//     Standard Inputs/MAIN.R2.In_From_HW/BYTE_[59] <-> Module 3 (Default IO)/Std. In (64 Bytes)/Input DWORD 14 @bit 16
//     Standard Inputs/MAIN.R2.In_From_HW/BYTE_[60] <-> Module 3 (Default IO)/Std. In (64 Bytes)/Input DWORD 14 @bit 24
//     Standard Inputs/MAIN.R2.In_From_HW/BYTE_[62] <-> Module 3 (Default IO)/Std. In (64 Bytes)/Input DWORD 15 @bit 8
//     Standard Inputs/MAIN.R2.In_From_HW/BYTE_[63] <-> Module 3 (Default IO)/Std. In (64 Bytes)/Input DWORD 15 @bit 16
//     Standard Inputs/MAIN.R2.In_From_HW/BYTE_[64] <-> Module 3 (Default IO)/Std. In (64 Bytes)/Input DWORD 15 @bit 24
//     Standard Inputs/MAIN.R2.In_From_HW/BYTE_[6] <-> Module 3 (Default IO)/Std. In (64 Bytes)/Input DWORD 1 @bit 8
//     Standard Inputs/MAIN.R2.In_From_HW/BYTE_[7] <-> Module 3 (Default IO)/Std. In (64 Bytes)/Input DWORD 1 @bit 16
//     Standard Inputs/MAIN.R2.In_From_HW/BYTE_[8] <-> Module 3 (Default IO)/Std. In (64 Bytes)/Input DWORD 1 @bit 24
//     Standard Inputs/MAIN.R2.In_From_HW/BYTE_[{1..61 step 4}] <-> Module 3 (Default IO)/Std. In (64 Bytes)/Input DWORD {0..15}  (16 links)
//     Standard Inputs/MAIN.R2.RT02/External_device_not_connected <-> Module 1 (Sync Inputs)/Compact/External device not connected
//     Standard Inputs/MAIN.R2.RT02/FSOE_Inputs_ConnID <-> Module 2 (Safety Data (8 Byte))/Inputs/FSOE/FSOE ConnID
//     Standard Inputs/MAIN.R2.RT02/FSOE_Inputs_Data_0 <-> Module 2 (Safety Data (8 Byte))/Inputs/FSOE/FSOE Data_0
//     Standard Inputs/MAIN.R2.RT02/FSOE_Inputs_Data_1 <-> Module 2 (Safety Data (8 Byte))/Inputs/FSOE/FSOE Data_1
//     Standard Inputs/MAIN.R2.RT02/FSOE_Inputs_Data_2 <-> Module 2 (Safety Data (8 Byte))/Inputs/FSOE/FSOE Data_2
//     Standard Inputs/MAIN.R2.RT02/FSOE_Inputs_Data_3 <-> Module 2 (Safety Data (8 Byte))/Inputs/FSOE/FSOE Data_3
//     Standard Inputs/MAIN.R2.RT02/InfoData/AdsAddr/netId <-> InfoData/AdsAddr/netId
//     Standard Inputs/MAIN.R2.RT02/InfoData/AdsAddr/port <-> InfoData/AdsAddr/port
//     Standard Inputs/MAIN.R2.RT02/InfoData/State <-> InfoData/State
//     Standard Inputs/MAIN.R2.RT02/TxPDO_State <-> Module 1 (Sync Inputs)/Compact/TxPDO state
//     Standard Inputs/MAIN.R2.RT02/TxPDO_Toogle <-> Module 1 (Sync Inputs)/Compact/TxPDO toggle
//     Standard Outputs/MAIN.R2.Out_To_HW/Byte_[10] <-> Module 3 (Default IO)/Std. Out (64 Bytes)/Output DWORD 2 @bit 8
//     Standard Outputs/MAIN.R2.Out_To_HW/Byte_[11] <-> Module 3 (Default IO)/Std. Out (64 Bytes)/Output DWORD 2 @bit 16
//     Standard Outputs/MAIN.R2.Out_To_HW/Byte_[12] <-> Module 3 (Default IO)/Std. Out (64 Bytes)/Output DWORD 2 @bit 24
//     Standard Outputs/MAIN.R2.Out_To_HW/Byte_[14] <-> Module 3 (Default IO)/Std. Out (64 Bytes)/Output DWORD 3 @bit 8
//     Standard Outputs/MAIN.R2.Out_To_HW/Byte_[15] <-> Module 3 (Default IO)/Std. Out (64 Bytes)/Output DWORD 3 @bit 16
//     Standard Outputs/MAIN.R2.Out_To_HW/Byte_[16] <-> Module 3 (Default IO)/Std. Out (64 Bytes)/Output DWORD 3 @bit 24
//     Standard Outputs/MAIN.R2.Out_To_HW/Byte_[18] <-> Module 3 (Default IO)/Std. Out (64 Bytes)/Output DWORD 4 @bit 8
//     Standard Outputs/MAIN.R2.Out_To_HW/Byte_[19] <-> Module 3 (Default IO)/Std. Out (64 Bytes)/Output DWORD 4 @bit 16
//     Standard Outputs/MAIN.R2.Out_To_HW/Byte_[20] <-> Module 3 (Default IO)/Std. Out (64 Bytes)/Output DWORD 4 @bit 24
//     Standard Outputs/MAIN.R2.Out_To_HW/Byte_[22] <-> Module 3 (Default IO)/Std. Out (64 Bytes)/Output DWORD 5 @bit 8
//     Standard Outputs/MAIN.R2.Out_To_HW/Byte_[23] <-> Module 3 (Default IO)/Std. Out (64 Bytes)/Output DWORD 5 @bit 16
//     Standard Outputs/MAIN.R2.Out_To_HW/Byte_[24] <-> Module 3 (Default IO)/Std. Out (64 Bytes)/Output DWORD 5 @bit 24
//     Standard Outputs/MAIN.R2.Out_To_HW/Byte_[26] <-> Module 3 (Default IO)/Std. Out (64 Bytes)/Output DWORD 6 @bit 8
//     Standard Outputs/MAIN.R2.Out_To_HW/Byte_[27] <-> Module 3 (Default IO)/Std. Out (64 Bytes)/Output DWORD 6 @bit 16
//     Standard Outputs/MAIN.R2.Out_To_HW/Byte_[28] <-> Module 3 (Default IO)/Std. Out (64 Bytes)/Output DWORD 6 @bit 24
//     Standard Outputs/MAIN.R2.Out_To_HW/Byte_[2] <-> Module 3 (Default IO)/Std. Out (64 Bytes)/Output DWORD 0 @bit 8
//     Standard Outputs/MAIN.R2.Out_To_HW/Byte_[30] <-> Module 3 (Default IO)/Std. Out (64 Bytes)/Output DWORD 7 @bit 8
//     Standard Outputs/MAIN.R2.Out_To_HW/Byte_[31] <-> Module 3 (Default IO)/Std. Out (64 Bytes)/Output DWORD 7 @bit 16
//     Standard Outputs/MAIN.R2.Out_To_HW/Byte_[32] <-> Module 3 (Default IO)/Std. Out (64 Bytes)/Output DWORD 7 @bit 24
//     Standard Outputs/MAIN.R2.Out_To_HW/Byte_[34] <-> Module 3 (Default IO)/Std. Out (64 Bytes)/Output DWORD 8 @bit 8
//     Standard Outputs/MAIN.R2.Out_To_HW/Byte_[35] <-> Module 3 (Default IO)/Std. Out (64 Bytes)/Output DWORD 8 @bit 16
//     Standard Outputs/MAIN.R2.Out_To_HW/Byte_[36] <-> Module 3 (Default IO)/Std. Out (64 Bytes)/Output DWORD 8 @bit 24
//     Standard Outputs/MAIN.R2.Out_To_HW/Byte_[38] <-> Module 3 (Default IO)/Std. Out (64 Bytes)/Output DWORD 9 @bit 8
//     Standard Outputs/MAIN.R2.Out_To_HW/Byte_[39] <-> Module 3 (Default IO)/Std. Out (64 Bytes)/Output DWORD 9 @bit 16
//     Standard Outputs/MAIN.R2.Out_To_HW/Byte_[3] <-> Module 3 (Default IO)/Std. Out (64 Bytes)/Output DWORD 0 @bit 16
//     Standard Outputs/MAIN.R2.Out_To_HW/Byte_[40] <-> Module 3 (Default IO)/Std. Out (64 Bytes)/Output DWORD 9 @bit 24
//     Standard Outputs/MAIN.R2.Out_To_HW/Byte_[42] <-> Module 3 (Default IO)/Std. Out (64 Bytes)/Output DWORD 10 @bit 8
//     Standard Outputs/MAIN.R2.Out_To_HW/Byte_[43] <-> Module 3 (Default IO)/Std. Out (64 Bytes)/Output DWORD 10 @bit 16
//     Standard Outputs/MAIN.R2.Out_To_HW/Byte_[44] <-> Module 3 (Default IO)/Std. Out (64 Bytes)/Output DWORD 10 @bit 24
//     Standard Outputs/MAIN.R2.Out_To_HW/Byte_[46] <-> Module 3 (Default IO)/Std. Out (64 Bytes)/Output DWORD 11 @bit 8
//     Standard Outputs/MAIN.R2.Out_To_HW/Byte_[47] <-> Module 3 (Default IO)/Std. Out (64 Bytes)/Output DWORD 11 @bit 16
//     Standard Outputs/MAIN.R2.Out_To_HW/Byte_[48] <-> Module 3 (Default IO)/Std. Out (64 Bytes)/Output DWORD 11 @bit 24
//     Standard Outputs/MAIN.R2.Out_To_HW/Byte_[4] <-> Module 3 (Default IO)/Std. Out (64 Bytes)/Output DWORD 0 @bit 24
//     Standard Outputs/MAIN.R2.Out_To_HW/Byte_[50] <-> Module 3 (Default IO)/Std. Out (64 Bytes)/Output DWORD 12 @bit 8
//     Standard Outputs/MAIN.R2.Out_To_HW/Byte_[51] <-> Module 3 (Default IO)/Std. Out (64 Bytes)/Output DWORD 12 @bit 16
//     Standard Outputs/MAIN.R2.Out_To_HW/Byte_[52] <-> Module 3 (Default IO)/Std. Out (64 Bytes)/Output DWORD 12 @bit 24
//     Standard Outputs/MAIN.R2.Out_To_HW/Byte_[54] <-> Module 3 (Default IO)/Std. Out (64 Bytes)/Output DWORD 13 @bit 8
//     Standard Outputs/MAIN.R2.Out_To_HW/Byte_[55] <-> Module 3 (Default IO)/Std. Out (64 Bytes)/Output DWORD 13 @bit 16
//     Standard Outputs/MAIN.R2.Out_To_HW/Byte_[56] <-> Module 3 (Default IO)/Std. Out (64 Bytes)/Output DWORD 13 @bit 24
//     Standard Outputs/MAIN.R2.Out_To_HW/Byte_[58] <-> Module 3 (Default IO)/Std. Out (64 Bytes)/Output DWORD 14 @bit 8
//     Standard Outputs/MAIN.R2.Out_To_HW/Byte_[59] <-> Module 3 (Default IO)/Std. Out (64 Bytes)/Output DWORD 14 @bit 16
//     Standard Outputs/MAIN.R2.Out_To_HW/Byte_[60] <-> Module 3 (Default IO)/Std. Out (64 Bytes)/Output DWORD 14 @bit 24
//     Standard Outputs/MAIN.R2.Out_To_HW/Byte_[62] <-> Module 3 (Default IO)/Std. Out (64 Bytes)/Output DWORD 15 @bit 8
//     Standard Outputs/MAIN.R2.Out_To_HW/Byte_[63] <-> Module 3 (Default IO)/Std. Out (64 Bytes)/Output DWORD 15 @bit 16
//     Standard Outputs/MAIN.R2.Out_To_HW/Byte_[64] <-> Module 3 (Default IO)/Std. Out (64 Bytes)/Output DWORD 15 @bit 24
//     Standard Outputs/MAIN.R2.Out_To_HW/Byte_[6] <-> Module 3 (Default IO)/Std. Out (64 Bytes)/Output DWORD 1 @bit 8
//     Standard Outputs/MAIN.R2.Out_To_HW/Byte_[7] <-> Module 3 (Default IO)/Std. Out (64 Bytes)/Output DWORD 1 @bit 16
//     Standard Outputs/MAIN.R2.Out_To_HW/Byte_[8] <-> Module 3 (Default IO)/Std. Out (64 Bytes)/Output DWORD 1 @bit 24
//     Standard Outputs/MAIN.R2.Out_To_HW/Byte_[{1..61 step 4}] <-> Module 3 (Default IO)/Std. Out (64 Bytes)/Output DWORD {0..15}  (16 links)
//   SODG11_SSCC610_2403701_PLC/SODG11_SSCC610_2403701_PLC Instance <-> EtherCAT Master (EtherCAT)/R2.T01 (EK1100)
//     Standard Inputs/MAIN.R2.T01/InfoData/State <-> InfoData/State
//   SODG11_SSCC610_2403701_PLC/SODG11_SSCC610_2403701_PLC Instance <-> EtherCAT Master (EtherCAT)/R2.T01 (EK1100)/R2.T02 (EL6900)
//     Standard Inputs/MAIN.R2.RT02/FSOE_Outputs_Data_0 @bit 1 <-> StandardInputs/Standard Out Var 14
//     Standard Inputs/MAIN.R2.RT02/FSOE_Outputs_Data_0 @bit 2 <-> StandardInputs/Standard Out Var 15
//     Standard Inputs/MAIN.R2.RT02/FSOE_Outputs_Data_2 @bit 1 <-> StandardInputs/Standard Out Var 18
//     Standard Inputs/MAIN.R2.RT02/FSOE_Outputs_Data_2 @bit 2 <-> StandardInputs/Standard Out Var 19
//     Standard Inputs/MAIN.R2.RT02/FSOE_Outputs_Data_2 @bit 3 <-> StandardInputs/Standard Out Var 20
//     Standard Inputs/MAIN.R2.RT02/FSOE_Outputs_Data_2 <-> StandardInputs/Standard Out Var 17
//     Standard Inputs/MAIN.R2.T02_STAT/Device_Info_Data/Project_CRC <-> Device Info Data/Project CRC
//     Standard Inputs/MAIN.R2.T02_STAT/FBs_FB_ERR <-> StandardInputs/Standard Out Var 16
//     Standard Inputs/MAIN.R2.T02_STAT/FBs_FB_ERR @bit 16 <-> StandardInputs/Standard Out Var 21
//     Standard Inputs/MAIN.R2.T02_STAT/FBs_FB_ERR @bit 29 <-> StandardInputs/Standard Out Var 22
//     Standard Inputs/MAIN.R2.T02_STAT/InfoData/AdsAddr/netId <-> InfoData/AdsAddr/netId
//     Standard Inputs/MAIN.R2.T02_STAT/InfoData/AdsAddr/port <-> InfoData/AdsAddr/port
//     Standard Inputs/MAIN.R2.T02_STAT/InfoData/State <-> InfoData/State
//     Standard Inputs/MAIN.R2.T02_STAT/SGs_COM_ERR @bit 1 <-> StandardInputs/Standard Out Var 12
//     Standard Inputs/MAIN.R2.T02_STAT/SGs_COM_ERR <-> StandardInputs/Standard Out Var 9
//     Standard Inputs/MAIN.R2.T02_STAT/SGs_FB_ERR @bit 1 <-> StandardInputs/Standard Out Var 11
//     Standard Inputs/MAIN.R2.T02_STAT/SGs_FB_ERR <-> StandardInputs/Standard Out Var 8
//     Standard Inputs/MAIN.R2.T02_STAT/SGs_OUT_ERR <-> StandardInputs/Standard Out Var 10
//     Standard Inputs/MAIN.R2.T02_STAT/SGs_OUT_ERR @bit 1 <-> StandardInputs/Standard Out Var 13
//     Standard Outputs/MAIN.R2.T02_CMD/FBs_ControlPowerPB <-> StandardOutputs/Standard In Var 7
//     Standard Outputs/MAIN.R2.T02_CMD/SGs_ERRAck <-> StandardOutputs/Standard In Var 4
//     Standard Outputs/MAIN.R2.T02_CMD/SGs_ERRAck <-> StandardOutputs/Standard In Var 6
//     Standard Outputs/MAIN.R2.T02_CMD/SGs_RUNSTOP <-> StandardOutputs/Standard In Var 3
//     Standard Outputs/MAIN.R2.T02_CMD/SGs_RUNSTOP <-> StandardOutputs/Standard In Var 5
//     Standard Outputs/MAIN.Safety_Zone_Test <-> StandardOutputs/Standard In Var 23
//   SODG11_SSCC610_2403701_PLC/SODG11_SSCC610_2403701_PLC Instance <-> EtherCAT Master (EtherCAT)/R2.T01 (EK1100)/R2.T03 (EL1904)
//     Standard Inputs/MAIN.R2.T03/I <-> Module 1 (FSOES)/TxPDO/FSOE/InputChannel1
//     Standard Inputs/MAIN.R2.T03/I @bit 1 <-> Module 1 (FSOES)/TxPDO/FSOE/InputChannel2
//     Standard Inputs/MAIN.R2.T03/I @bit 2 <-> Module 1 (FSOES)/TxPDO/FSOE/InputChannel3
//     Standard Inputs/MAIN.R2.T03/I @bit 3 <-> Module 1 (FSOES)/TxPDO/FSOE/InputChannel4
//     Standard Inputs/MAIN.R2.T03/InfoData/State <-> InfoData/State
//   SODG11_SSCC610_2403701_PLC/SODG11_SSCC610_2403701_PLC Instance <-> EtherCAT Master (EtherCAT)/R2.T01 (EK1100)/R2.T04 (EK1122)
//     Standard Inputs/MAIN.R2.T04/InfoData/State <-> InfoData/State
//   SODG11_SSCC610_2403701_PLC/SODG11_SSCC610_2403701_PLC Instance <-> EtherCAT Master (EtherCAT)/R2.T01 (EK1100)/R2.T04 (EK1122)/R2.Reamer[1].N01 (EP1008-0002)
//     Standard Inputs/MAIN.R2.Reamer[1].N01/I <-> Channel 1/Input
//     Standard Inputs/MAIN.R2.Reamer[1].N01/I @bit 1 <-> Channel 2/Input
//     Standard Inputs/MAIN.R2.Reamer[1].N01/I @bit 2 <-> Channel 3/Input
//     Standard Inputs/MAIN.R2.Reamer[1].N01/I @bit 3 <-> Channel 4/Input
//     Standard Inputs/MAIN.R2.Reamer[1].N01/I @bit 4 <-> Channel 5/Input
//     Standard Inputs/MAIN.R2.Reamer[1].N01/I @bit 5 <-> Channel 6/Input
//     Standard Inputs/MAIN.R2.Reamer[1].N01/I @bit 6 <-> Channel 7/Input
//     Standard Inputs/MAIN.R2.Reamer[1].N01/I @bit 7 <-> Channel 8/Input
//     Standard Inputs/MAIN.R2.Reamer[1].N01/InfoData/State <-> InfoData/State
//     Standard Inputs/MAIN.R2.Reamer[1].N01/Wc_State <-> WcState/WcState
//   SODG11_SSCC610_2403701_PLC/SODG11_SSCC610_2403701_PLC Instance <-> EtherCAT Master (EtherCAT)/R2.T01 (EK1100)/R2.T04 (EK1122)/R2.Reamer[1].N30 (EP2028-0002)
//     Standard Inputs/MAIN.R2.Reamer[1].N30_STAT/InfoData/State <-> InfoData/State
//     Standard Outputs/MAIN.R2.Reamer[1].N30/Q <-> Channel 1/Output
//     Standard Outputs/MAIN.R2.Reamer[1].N30/Q @bit {1..7} <-> Channel {2..8}/Output  (7 links)
//   SODG11_SSCC610_2403701_PLC/SODG11_SSCC610_2403701_PLC Instance <-> EtherCAT Master (EtherCAT)/R3.RT02 (EL6695-1001)
//     Standard Inputs/MAIN.R3.In_From_HW/BYTE_[10] <-> Module 3 (Default IO)/Std. In (64 Bytes)/Input DWORD 2 @bit 8
//     Standard Inputs/MAIN.R3.In_From_HW/BYTE_[11] <-> Module 3 (Default IO)/Std. In (64 Bytes)/Input DWORD 2 @bit 16
//     Standard Inputs/MAIN.R3.In_From_HW/BYTE_[12] <-> Module 3 (Default IO)/Std. In (64 Bytes)/Input DWORD 2 @bit 24
//     Standard Inputs/MAIN.R3.In_From_HW/BYTE_[14] <-> Module 3 (Default IO)/Std. In (64 Bytes)/Input DWORD 3 @bit 8
//     Standard Inputs/MAIN.R3.In_From_HW/BYTE_[15] <-> Module 3 (Default IO)/Std. In (64 Bytes)/Input DWORD 3 @bit 16
//     Standard Inputs/MAIN.R3.In_From_HW/BYTE_[16] <-> Module 3 (Default IO)/Std. In (64 Bytes)/Input DWORD 3 @bit 24
//     Standard Inputs/MAIN.R3.In_From_HW/BYTE_[18] <-> Module 3 (Default IO)/Std. In (64 Bytes)/Input DWORD 4 @bit 8
//     Standard Inputs/MAIN.R3.In_From_HW/BYTE_[19] <-> Module 3 (Default IO)/Std. In (64 Bytes)/Input DWORD 4 @bit 16
//     Standard Inputs/MAIN.R3.In_From_HW/BYTE_[20] <-> Module 3 (Default IO)/Std. In (64 Bytes)/Input DWORD 4 @bit 24
//     Standard Inputs/MAIN.R3.In_From_HW/BYTE_[22] <-> Module 3 (Default IO)/Std. In (64 Bytes)/Input DWORD 5 @bit 8
//     Standard Inputs/MAIN.R3.In_From_HW/BYTE_[23] <-> Module 3 (Default IO)/Std. In (64 Bytes)/Input DWORD 5 @bit 16
//     Standard Inputs/MAIN.R3.In_From_HW/BYTE_[24] <-> Module 3 (Default IO)/Std. In (64 Bytes)/Input DWORD 5 @bit 24
//     Standard Inputs/MAIN.R3.In_From_HW/BYTE_[26] <-> Module 3 (Default IO)/Std. In (64 Bytes)/Input DWORD 6 @bit 8
//     Standard Inputs/MAIN.R3.In_From_HW/BYTE_[27] <-> Module 3 (Default IO)/Std. In (64 Bytes)/Input DWORD 6 @bit 16
//     Standard Inputs/MAIN.R3.In_From_HW/BYTE_[28] <-> Module 3 (Default IO)/Std. In (64 Bytes)/Input DWORD 6 @bit 24
//     Standard Inputs/MAIN.R3.In_From_HW/BYTE_[2] <-> Module 3 (Default IO)/Std. In (64 Bytes)/Input DWORD 0 @bit 8
//     Standard Inputs/MAIN.R3.In_From_HW/BYTE_[30] <-> Module 3 (Default IO)/Std. In (64 Bytes)/Input DWORD 7 @bit 8
//     Standard Inputs/MAIN.R3.In_From_HW/BYTE_[31] <-> Module 3 (Default IO)/Std. In (64 Bytes)/Input DWORD 7 @bit 16
//     Standard Inputs/MAIN.R3.In_From_HW/BYTE_[32] <-> Module 3 (Default IO)/Std. In (64 Bytes)/Input DWORD 7 @bit 24
//     Standard Inputs/MAIN.R3.In_From_HW/BYTE_[34] <-> Module 3 (Default IO)/Std. In (64 Bytes)/Input DWORD 8 @bit 8
//     Standard Inputs/MAIN.R3.In_From_HW/BYTE_[35] <-> Module 3 (Default IO)/Std. In (64 Bytes)/Input DWORD 8 @bit 16
//     Standard Inputs/MAIN.R3.In_From_HW/BYTE_[36] <-> Module 3 (Default IO)/Std. In (64 Bytes)/Input DWORD 8 @bit 24
//     Standard Inputs/MAIN.R3.In_From_HW/BYTE_[38] <-> Module 3 (Default IO)/Std. In (64 Bytes)/Input DWORD 9 @bit 8
//     Standard Inputs/MAIN.R3.In_From_HW/BYTE_[39] <-> Module 3 (Default IO)/Std. In (64 Bytes)/Input DWORD 9 @bit 16
//     Standard Inputs/MAIN.R3.In_From_HW/BYTE_[3] <-> Module 3 (Default IO)/Std. In (64 Bytes)/Input DWORD 0 @bit 16
//     Standard Inputs/MAIN.R3.In_From_HW/BYTE_[40] <-> Module 3 (Default IO)/Std. In (64 Bytes)/Input DWORD 9 @bit 24
//     Standard Inputs/MAIN.R3.In_From_HW/BYTE_[42] <-> Module 3 (Default IO)/Std. In (64 Bytes)/Input DWORD 10 @bit 8
//     Standard Inputs/MAIN.R3.In_From_HW/BYTE_[43] <-> Module 3 (Default IO)/Std. In (64 Bytes)/Input DWORD 10 @bit 16
//     Standard Inputs/MAIN.R3.In_From_HW/BYTE_[44] <-> Module 3 (Default IO)/Std. In (64 Bytes)/Input DWORD 10 @bit 24
//     Standard Inputs/MAIN.R3.In_From_HW/BYTE_[46] <-> Module 3 (Default IO)/Std. In (64 Bytes)/Input DWORD 11 @bit 8
//     Standard Inputs/MAIN.R3.In_From_HW/BYTE_[47] <-> Module 3 (Default IO)/Std. In (64 Bytes)/Input DWORD 11 @bit 16
//     Standard Inputs/MAIN.R3.In_From_HW/BYTE_[48] <-> Module 3 (Default IO)/Std. In (64 Bytes)/Input DWORD 11 @bit 24
//     Standard Inputs/MAIN.R3.In_From_HW/BYTE_[4] <-> Module 3 (Default IO)/Std. In (64 Bytes)/Input DWORD 0 @bit 24
//     Standard Inputs/MAIN.R3.In_From_HW/BYTE_[50] <-> Module 3 (Default IO)/Std. In (64 Bytes)/Input DWORD 12 @bit 8
//     Standard Inputs/MAIN.R3.In_From_HW/BYTE_[51] <-> Module 3 (Default IO)/Std. In (64 Bytes)/Input DWORD 12 @bit 16
//     Standard Inputs/MAIN.R3.In_From_HW/BYTE_[52] <-> Module 3 (Default IO)/Std. In (64 Bytes)/Input DWORD 12 @bit 24
//     Standard Inputs/MAIN.R3.In_From_HW/BYTE_[54] <-> Module 3 (Default IO)/Std. In (64 Bytes)/Input DWORD 13 @bit 8
//     Standard Inputs/MAIN.R3.In_From_HW/BYTE_[55] <-> Module 3 (Default IO)/Std. In (64 Bytes)/Input DWORD 13 @bit 16
//     Standard Inputs/MAIN.R3.In_From_HW/BYTE_[56] <-> Module 3 (Default IO)/Std. In (64 Bytes)/Input DWORD 13 @bit 24
//     Standard Inputs/MAIN.R3.In_From_HW/BYTE_[58] <-> Module 3 (Default IO)/Std. In (64 Bytes)/Input DWORD 14 @bit 8
//     Standard Inputs/MAIN.R3.In_From_HW/BYTE_[59] <-> Module 3 (Default IO)/Std. In (64 Bytes)/Input DWORD 14 @bit 16
//     Standard Inputs/MAIN.R3.In_From_HW/BYTE_[60] <-> Module 3 (Default IO)/Std. In (64 Bytes)/Input DWORD 14 @bit 24
//     Standard Inputs/MAIN.R3.In_From_HW/BYTE_[62] <-> Module 3 (Default IO)/Std. In (64 Bytes)/Input DWORD 15 @bit 8
//     Standard Inputs/MAIN.R3.In_From_HW/BYTE_[63] <-> Module 3 (Default IO)/Std. In (64 Bytes)/Input DWORD 15 @bit 16
//     Standard Inputs/MAIN.R3.In_From_HW/BYTE_[64] <-> Module 3 (Default IO)/Std. In (64 Bytes)/Input DWORD 15 @bit 24
//     Standard Inputs/MAIN.R3.In_From_HW/BYTE_[6] <-> Module 3 (Default IO)/Std. In (64 Bytes)/Input DWORD 1 @bit 8
//     Standard Inputs/MAIN.R3.In_From_HW/BYTE_[7] <-> Module 3 (Default IO)/Std. In (64 Bytes)/Input DWORD 1 @bit 16
//     Standard Inputs/MAIN.R3.In_From_HW/BYTE_[8] <-> Module 3 (Default IO)/Std. In (64 Bytes)/Input DWORD 1 @bit 24
//     Standard Inputs/MAIN.R3.In_From_HW/BYTE_[{1..61 step 4}] <-> Module 3 (Default IO)/Std. In (64 Bytes)/Input DWORD {0..15}  (16 links)
//     Standard Inputs/MAIN.R3.RT02/External_device_not_connected <-> Module 1 (Sync Inputs)/Compact/External device not connected
//     Standard Inputs/MAIN.R3.RT02/FSOE_Inputs_ConnID <-> Module 2 (Safety Data (8 Byte))/Inputs/FSOE/FSOE ConnID
//     Standard Inputs/MAIN.R3.RT02/FSOE_Inputs_Data_0 <-> Module 2 (Safety Data (8 Byte))/Inputs/FSOE/FSOE Data_0
//     Standard Inputs/MAIN.R3.RT02/FSOE_Inputs_Data_1 <-> Module 2 (Safety Data (8 Byte))/Inputs/FSOE/FSOE Data_1
//     Standard Inputs/MAIN.R3.RT02/FSOE_Inputs_Data_2 <-> Module 2 (Safety Data (8 Byte))/Inputs/FSOE/FSOE Data_2
//     Standard Inputs/MAIN.R3.RT02/FSOE_Inputs_Data_3 <-> Module 2 (Safety Data (8 Byte))/Inputs/FSOE/FSOE Data_3
//     Standard Inputs/MAIN.R3.RT02/InfoData/AdsAddr/netId <-> InfoData/AdsAddr/netId
//     Standard Inputs/MAIN.R3.RT02/InfoData/AdsAddr/port <-> InfoData/AdsAddr/port
//     Standard Inputs/MAIN.R3.RT02/InfoData/State <-> InfoData/State
//     Standard Inputs/MAIN.R3.RT02/TxPDO_State <-> Module 1 (Sync Inputs)/Compact/TxPDO state
//     Standard Inputs/MAIN.R3.RT02/TxPDO_Toogle <-> Module 1 (Sync Inputs)/Compact/TxPDO toggle
//     Standard Outputs/MAIN.R3.Out_To_HW/Byte_[10] <-> Module 3 (Default IO)/Std. Out (64 Bytes)/Output DWORD 2 @bit 8
//     Standard Outputs/MAIN.R3.Out_To_HW/Byte_[11] <-> Module 3 (Default IO)/Std. Out (64 Bytes)/Output DWORD 2 @bit 16
//     Standard Outputs/MAIN.R3.Out_To_HW/Byte_[12] <-> Module 3 (Default IO)/Std. Out (64 Bytes)/Output DWORD 2 @bit 24
//     Standard Outputs/MAIN.R3.Out_To_HW/Byte_[14] <-> Module 3 (Default IO)/Std. Out (64 Bytes)/Output DWORD 3 @bit 8
//     Standard Outputs/MAIN.R3.Out_To_HW/Byte_[15] <-> Module 3 (Default IO)/Std. Out (64 Bytes)/Output DWORD 3 @bit 16
//     Standard Outputs/MAIN.R3.Out_To_HW/Byte_[16] <-> Module 3 (Default IO)/Std. Out (64 Bytes)/Output DWORD 3 @bit 24
//     Standard Outputs/MAIN.R3.Out_To_HW/Byte_[18] <-> Module 3 (Default IO)/Std. Out (64 Bytes)/Output DWORD 4 @bit 8
//     Standard Outputs/MAIN.R3.Out_To_HW/Byte_[19] <-> Module 3 (Default IO)/Std. Out (64 Bytes)/Output DWORD 4 @bit 16
//     Standard Outputs/MAIN.R3.Out_To_HW/Byte_[20] <-> Module 3 (Default IO)/Std. Out (64 Bytes)/Output DWORD 4 @bit 24
//     Standard Outputs/MAIN.R3.Out_To_HW/Byte_[22] <-> Module 3 (Default IO)/Std. Out (64 Bytes)/Output DWORD 5 @bit 8
//     Standard Outputs/MAIN.R3.Out_To_HW/Byte_[23] <-> Module 3 (Default IO)/Std. Out (64 Bytes)/Output DWORD 5 @bit 16
//     Standard Outputs/MAIN.R3.Out_To_HW/Byte_[24] <-> Module 3 (Default IO)/Std. Out (64 Bytes)/Output DWORD 5 @bit 24
//     Standard Outputs/MAIN.R3.Out_To_HW/Byte_[26] <-> Module 3 (Default IO)/Std. Out (64 Bytes)/Output DWORD 6 @bit 8
//     Standard Outputs/MAIN.R3.Out_To_HW/Byte_[27] <-> Module 3 (Default IO)/Std. Out (64 Bytes)/Output DWORD 6 @bit 16
//     Standard Outputs/MAIN.R3.Out_To_HW/Byte_[28] <-> Module 3 (Default IO)/Std. Out (64 Bytes)/Output DWORD 6 @bit 24
//     Standard Outputs/MAIN.R3.Out_To_HW/Byte_[2] <-> Module 3 (Default IO)/Std. Out (64 Bytes)/Output DWORD 0 @bit 8
//     Standard Outputs/MAIN.R3.Out_To_HW/Byte_[30] <-> Module 3 (Default IO)/Std. Out (64 Bytes)/Output DWORD 7 @bit 8
//     Standard Outputs/MAIN.R3.Out_To_HW/Byte_[31] <-> Module 3 (Default IO)/Std. Out (64 Bytes)/Output DWORD 7 @bit 16
//     Standard Outputs/MAIN.R3.Out_To_HW/Byte_[32] <-> Module 3 (Default IO)/Std. Out (64 Bytes)/Output DWORD 7 @bit 24
//     Standard Outputs/MAIN.R3.Out_To_HW/Byte_[34] <-> Module 3 (Default IO)/Std. Out (64 Bytes)/Output DWORD 8 @bit 8
//     Standard Outputs/MAIN.R3.Out_To_HW/Byte_[35] <-> Module 3 (Default IO)/Std. Out (64 Bytes)/Output DWORD 8 @bit 16
//     Standard Outputs/MAIN.R3.Out_To_HW/Byte_[36] <-> Module 3 (Default IO)/Std. Out (64 Bytes)/Output DWORD 8 @bit 24
//     Standard Outputs/MAIN.R3.Out_To_HW/Byte_[38] <-> Module 3 (Default IO)/Std. Out (64 Bytes)/Output DWORD 9 @bit 8
//     Standard Outputs/MAIN.R3.Out_To_HW/Byte_[39] <-> Module 3 (Default IO)/Std. Out (64 Bytes)/Output DWORD 9 @bit 16
//     Standard Outputs/MAIN.R3.Out_To_HW/Byte_[3] <-> Module 3 (Default IO)/Std. Out (64 Bytes)/Output DWORD 0 @bit 16
//     Standard Outputs/MAIN.R3.Out_To_HW/Byte_[40] <-> Module 3 (Default IO)/Std. Out (64 Bytes)/Output DWORD 9 @bit 24
//     Standard Outputs/MAIN.R3.Out_To_HW/Byte_[42] <-> Module 3 (Default IO)/Std. Out (64 Bytes)/Output DWORD 10 @bit 8
//     Standard Outputs/MAIN.R3.Out_To_HW/Byte_[43] <-> Module 3 (Default IO)/Std. Out (64 Bytes)/Output DWORD 10 @bit 16
//     Standard Outputs/MAIN.R3.Out_To_HW/Byte_[44] <-> Module 3 (Default IO)/Std. Out (64 Bytes)/Output DWORD 10 @bit 24
//     Standard Outputs/MAIN.R3.Out_To_HW/Byte_[46] <-> Module 3 (Default IO)/Std. Out (64 Bytes)/Output DWORD 11 @bit 8
//     Standard Outputs/MAIN.R3.Out_To_HW/Byte_[47] <-> Module 3 (Default IO)/Std. Out (64 Bytes)/Output DWORD 11 @bit 16
//     Standard Outputs/MAIN.R3.Out_To_HW/Byte_[48] <-> Module 3 (Default IO)/Std. Out (64 Bytes)/Output DWORD 11 @bit 24
//     Standard Outputs/MAIN.R3.Out_To_HW/Byte_[4] <-> Module 3 (Default IO)/Std. Out (64 Bytes)/Output DWORD 0 @bit 24
//     Standard Outputs/MAIN.R3.Out_To_HW/Byte_[50] <-> Module 3 (Default IO)/Std. Out (64 Bytes)/Output DWORD 12 @bit 8
//     Standard Outputs/MAIN.R3.Out_To_HW/Byte_[51] <-> Module 3 (Default IO)/Std. Out (64 Bytes)/Output DWORD 12 @bit 16
//     Standard Outputs/MAIN.R3.Out_To_HW/Byte_[52] <-> Module 3 (Default IO)/Std. Out (64 Bytes)/Output DWORD 12 @bit 24
//     Standard Outputs/MAIN.R3.Out_To_HW/Byte_[54] <-> Module 3 (Default IO)/Std. Out (64 Bytes)/Output DWORD 13 @bit 8
//     Standard Outputs/MAIN.R3.Out_To_HW/Byte_[55] <-> Module 3 (Default IO)/Std. Out (64 Bytes)/Output DWORD 13 @bit 16
//     Standard Outputs/MAIN.R3.Out_To_HW/Byte_[56] <-> Module 3 (Default IO)/Std. Out (64 Bytes)/Output DWORD 13 @bit 24
//     Standard Outputs/MAIN.R3.Out_To_HW/Byte_[58] <-> Module 3 (Default IO)/Std. Out (64 Bytes)/Output DWORD 14 @bit 8
//     Standard Outputs/MAIN.R3.Out_To_HW/Byte_[59] <-> Module 3 (Default IO)/Std. Out (64 Bytes)/Output DWORD 14 @bit 16
//     Standard Outputs/MAIN.R3.Out_To_HW/Byte_[60] <-> Module 3 (Default IO)/Std. Out (64 Bytes)/Output DWORD 14 @bit 24
//     Standard Outputs/MAIN.R3.Out_To_HW/Byte_[62] <-> Module 3 (Default IO)/Std. Out (64 Bytes)/Output DWORD 15 @bit 8
//     Standard Outputs/MAIN.R3.Out_To_HW/Byte_[63] <-> Module 3 (Default IO)/Std. Out (64 Bytes)/Output DWORD 15 @bit 16
//     Standard Outputs/MAIN.R3.Out_To_HW/Byte_[64] <-> Module 3 (Default IO)/Std. Out (64 Bytes)/Output DWORD 15 @bit 24
//     Standard Outputs/MAIN.R3.Out_To_HW/Byte_[6] <-> Module 3 (Default IO)/Std. Out (64 Bytes)/Output DWORD 1 @bit 8
//     Standard Outputs/MAIN.R3.Out_To_HW/Byte_[7] <-> Module 3 (Default IO)/Std. Out (64 Bytes)/Output DWORD 1 @bit 16
//     Standard Outputs/MAIN.R3.Out_To_HW/Byte_[8] <-> Module 3 (Default IO)/Std. Out (64 Bytes)/Output DWORD 1 @bit 24
//     Standard Outputs/MAIN.R3.Out_To_HW/Byte_[{1..61 step 4}] <-> Module 3 (Default IO)/Std. Out (64 Bytes)/Output DWORD {0..15}  (16 links)
//   SODG11_SSCC610_2403701_PLC/SODG11_SSCC610_2403701_PLC Instance <-> EtherCAT Master (EtherCAT)/R3.T01 (EK1100)
//     Standard Inputs/MAIN.R3.T01/InfoData/State <-> InfoData/State
//   SODG11_SSCC610_2403701_PLC/SODG11_SSCC610_2403701_PLC Instance <-> EtherCAT Master (EtherCAT)/R3.T01 (EK1100)/R3.T02 (EL6900)
//     Standard Inputs/MAIN.R3.RT02/FSOE_Outputs_Data_0 @bit 1 <-> StandardInputs/Standard Out Var 14
//     Standard Inputs/MAIN.R3.RT02/FSOE_Outputs_Data_0 @bit 2 <-> StandardInputs/Standard Out Var 15
//     Standard Inputs/MAIN.R3.RT02/FSOE_Outputs_Data_2 @bit 1 <-> StandardInputs/Standard Out Var 18
//     Standard Inputs/MAIN.R3.RT02/FSOE_Outputs_Data_2 <-> StandardInputs/Standard Out Var 17
//     Standard Inputs/MAIN.R3.T02_STAT/Device_Info_Data/Project_CRC <-> Device Info Data/Project CRC
//     Standard Inputs/MAIN.R3.T02_STAT/FBs_FB_ERR <-> StandardInputs/Standard Out Var 16
//     Standard Inputs/MAIN.R3.T02_STAT/FBs_FB_ERR @bit 16 <-> StandardInputs/Standard Out Var 19
//     Standard Inputs/MAIN.R3.T02_STAT/FBs_FB_ERR @bit 29 <-> StandardInputs/Standard Out Var 20
//     Standard Inputs/MAIN.R3.T02_STAT/InfoData/AdsAddr/netId <-> InfoData/AdsAddr/netId
//     Standard Inputs/MAIN.R3.T02_STAT/InfoData/AdsAddr/port <-> InfoData/AdsAddr/port
//     Standard Inputs/MAIN.R3.T02_STAT/InfoData/State <-> InfoData/State
//     Standard Inputs/MAIN.R3.T02_STAT/SGs_COM_ERR @bit 1 <-> StandardInputs/Standard Out Var 12
//     Standard Inputs/MAIN.R3.T02_STAT/SGs_COM_ERR <-> StandardInputs/Standard Out Var 9
//     Standard Inputs/MAIN.R3.T02_STAT/SGs_FB_ERR @bit 1 <-> StandardInputs/Standard Out Var 11
//     Standard Inputs/MAIN.R3.T02_STAT/SGs_FB_ERR <-> StandardInputs/Standard Out Var 8
//     Standard Inputs/MAIN.R3.T02_STAT/SGs_OUT_ERR <-> StandardInputs/Standard Out Var 10
//     Standard Inputs/MAIN.R3.T02_STAT/SGs_OUT_ERR @bit 1 <-> StandardInputs/Standard Out Var 13
//     Standard Outputs/MAIN.R3.T02_CMD/FBs_ControlPowerPB <-> StandardOutputs/Standard In Var 7
//     Standard Outputs/MAIN.R3.T02_CMD/SGs_ERRAck <-> StandardOutputs/Standard In Var 4
//     Standard Outputs/MAIN.R3.T02_CMD/SGs_ERRAck <-> StandardOutputs/Standard In Var 6
//     Standard Outputs/MAIN.R3.T02_CMD/SGs_RUNSTOP <-> StandardOutputs/Standard In Var 3
//     Standard Outputs/MAIN.R3.T02_CMD/SGs_RUNSTOP <-> StandardOutputs/Standard In Var 5
//     Standard Outputs/MAIN.Safety_Zone_Test <-> StandardOutputs/Standard In Var 21
//   SODG11_SSCC610_2403701_PLC/SODG11_SSCC610_2403701_PLC Instance <-> EtherCAT Master (EtherCAT)/R3.T01 (EK1100)/R3.T03 (EL1904)
//     Standard Inputs/MAIN.R3.T03/I <-> Module 1 (FSOES)/TxPDO/FSOE/InputChannel1
//     Standard Inputs/MAIN.R3.T03/I @bit 1 <-> Module 1 (FSOES)/TxPDO/FSOE/InputChannel2
//     Standard Inputs/MAIN.R3.T03/I @bit 2 <-> Module 1 (FSOES)/TxPDO/FSOE/InputChannel3
//     Standard Inputs/MAIN.R3.T03/I @bit 3 <-> Module 1 (FSOES)/TxPDO/FSOE/InputChannel4
//     Standard Inputs/MAIN.R3.T03/InfoData/State <-> InfoData/State
//   SODG11_SSCC610_2403701_PLC/SODG11_SSCC610_2403701_PLC Instance <-> EtherCAT Master (EtherCAT)/R3.T01 (EK1100)/R3.T04 (EK1122)
//     Standard Inputs/MAIN.R3.T04/InfoData/State <-> InfoData/State
//   SODG11_SSCC610_2403701_PLC/SODG11_SSCC610_2403701_PLC Instance <-> EtherCAT Master (EtherCAT)/R3.T01 (EK1100)/R3.T04 (EK1122)/R3.Reamer[1].N01 (EP1008-0002)
//     Standard Inputs/MAIN.R3.Reamer[1].N01/I <-> Channel 1/Input
//     Standard Inputs/MAIN.R3.Reamer[1].N01/I @bit 1 <-> Channel 2/Input
//     Standard Inputs/MAIN.R3.Reamer[1].N01/I @bit 2 <-> Channel 3/Input
//     Standard Inputs/MAIN.R3.Reamer[1].N01/I @bit 3 <-> Channel 4/Input
//     Standard Inputs/MAIN.R3.Reamer[1].N01/I @bit 4 <-> Channel 5/Input
//     Standard Inputs/MAIN.R3.Reamer[1].N01/I @bit 5 <-> Channel 6/Input
//     Standard Inputs/MAIN.R3.Reamer[1].N01/I @bit 6 <-> Channel 7/Input
//     Standard Inputs/MAIN.R3.Reamer[1].N01/I @bit 7 <-> Channel 8/Input
//     Standard Inputs/MAIN.R3.Reamer[1].N01/InfoData/State <-> InfoData/State
//     Standard Inputs/MAIN.R3.Reamer[1].N01/Wc_State <-> WcState/WcState
//   SODG11_SSCC610_2403701_PLC/SODG11_SSCC610_2403701_PLC Instance <-> EtherCAT Master (EtherCAT)/R3.T01 (EK1100)/R3.T04 (EK1122)/R3.Reamer[1].N30 (EP2028-0002)
//     Standard Inputs/MAIN.R3.Reamer[1].N30_STAT/InfoData/State <-> InfoData/State
//     Standard Outputs/MAIN.R3.Reamer[1].N30/Q <-> Channel 1/Output
//     Standard Outputs/MAIN.R3.Reamer[1].N30/Q @bit {1..7} <-> Channel {2..8}/Output  (7 links)
//   SODG11_SSCC610_2403701_PLC/SODG11_SSCC610_2403701_PLC Instance <-> EtherCAT Master (EtherCAT)/R4.RT02 (EL6695-1001)
//     Standard Inputs/MAIN.R4.In_From_HW/BYTE_[10] <-> Module 3 (Default IO)/Std. In (64 Bytes)/Input DWORD 2 @bit 8
//     Standard Inputs/MAIN.R4.In_From_HW/BYTE_[11] <-> Module 3 (Default IO)/Std. In (64 Bytes)/Input DWORD 2 @bit 16
//     Standard Inputs/MAIN.R4.In_From_HW/BYTE_[12] <-> Module 3 (Default IO)/Std. In (64 Bytes)/Input DWORD 2 @bit 24
//     Standard Inputs/MAIN.R4.In_From_HW/BYTE_[14] <-> Module 3 (Default IO)/Std. In (64 Bytes)/Input DWORD 3 @bit 8
//     Standard Inputs/MAIN.R4.In_From_HW/BYTE_[15] <-> Module 3 (Default IO)/Std. In (64 Bytes)/Input DWORD 3 @bit 16
//     Standard Inputs/MAIN.R4.In_From_HW/BYTE_[16] <-> Module 3 (Default IO)/Std. In (64 Bytes)/Input DWORD 3 @bit 24
//     Standard Inputs/MAIN.R4.In_From_HW/BYTE_[18] <-> Module 3 (Default IO)/Std. In (64 Bytes)/Input DWORD 4 @bit 8
//     Standard Inputs/MAIN.R4.In_From_HW/BYTE_[19] <-> Module 3 (Default IO)/Std. In (64 Bytes)/Input DWORD 4 @bit 16
//     Standard Inputs/MAIN.R4.In_From_HW/BYTE_[20] <-> Module 3 (Default IO)/Std. In (64 Bytes)/Input DWORD 4 @bit 24
//     Standard Inputs/MAIN.R4.In_From_HW/BYTE_[22] <-> Module 3 (Default IO)/Std. In (64 Bytes)/Input DWORD 5 @bit 8
//     Standard Inputs/MAIN.R4.In_From_HW/BYTE_[23] <-> Module 3 (Default IO)/Std. In (64 Bytes)/Input DWORD 5 @bit 16
//     Standard Inputs/MAIN.R4.In_From_HW/BYTE_[24] <-> Module 3 (Default IO)/Std. In (64 Bytes)/Input DWORD 5 @bit 24
//     Standard Inputs/MAIN.R4.In_From_HW/BYTE_[26] <-> Module 3 (Default IO)/Std. In (64 Bytes)/Input DWORD 6 @bit 8
//     Standard Inputs/MAIN.R4.In_From_HW/BYTE_[27] <-> Module 3 (Default IO)/Std. In (64 Bytes)/Input DWORD 6 @bit 16
//     Standard Inputs/MAIN.R4.In_From_HW/BYTE_[28] <-> Module 3 (Default IO)/Std. In (64 Bytes)/Input DWORD 6 @bit 24
//     Standard Inputs/MAIN.R4.In_From_HW/BYTE_[2] <-> Module 3 (Default IO)/Std. In (64 Bytes)/Input DWORD 0 @bit 8
//     Standard Inputs/MAIN.R4.In_From_HW/BYTE_[30] <-> Module 3 (Default IO)/Std. In (64 Bytes)/Input DWORD 7 @bit 8
//     Standard Inputs/MAIN.R4.In_From_HW/BYTE_[31] <-> Module 3 (Default IO)/Std. In (64 Bytes)/Input DWORD 7 @bit 16
//     Standard Inputs/MAIN.R4.In_From_HW/BYTE_[32] <-> Module 3 (Default IO)/Std. In (64 Bytes)/Input DWORD 7 @bit 24
//     Standard Inputs/MAIN.R4.In_From_HW/BYTE_[34] <-> Module 3 (Default IO)/Std. In (64 Bytes)/Input DWORD 8 @bit 8
//     Standard Inputs/MAIN.R4.In_From_HW/BYTE_[35] <-> Module 3 (Default IO)/Std. In (64 Bytes)/Input DWORD 8 @bit 16
//     Standard Inputs/MAIN.R4.In_From_HW/BYTE_[36] <-> Module 3 (Default IO)/Std. In (64 Bytes)/Input DWORD 8 @bit 24
//     Standard Inputs/MAIN.R4.In_From_HW/BYTE_[38] <-> Module 3 (Default IO)/Std. In (64 Bytes)/Input DWORD 9 @bit 8
//     Standard Inputs/MAIN.R4.In_From_HW/BYTE_[39] <-> Module 3 (Default IO)/Std. In (64 Bytes)/Input DWORD 9 @bit 16
//     Standard Inputs/MAIN.R4.In_From_HW/BYTE_[3] <-> Module 3 (Default IO)/Std. In (64 Bytes)/Input DWORD 0 @bit 16
//     Standard Inputs/MAIN.R4.In_From_HW/BYTE_[40] <-> Module 3 (Default IO)/Std. In (64 Bytes)/Input DWORD 9 @bit 24
//     Standard Inputs/MAIN.R4.In_From_HW/BYTE_[42] <-> Module 3 (Default IO)/Std. In (64 Bytes)/Input DWORD 10 @bit 8
//     Standard Inputs/MAIN.R4.In_From_HW/BYTE_[43] <-> Module 3 (Default IO)/Std. In (64 Bytes)/Input DWORD 10 @bit 16
//     Standard Inputs/MAIN.R4.In_From_HW/BYTE_[44] <-> Module 3 (Default IO)/Std. In (64 Bytes)/Input DWORD 10 @bit 24
//     Standard Inputs/MAIN.R4.In_From_HW/BYTE_[46] <-> Module 3 (Default IO)/Std. In (64 Bytes)/Input DWORD 11 @bit 8
//     Standard Inputs/MAIN.R4.In_From_HW/BYTE_[47] <-> Module 3 (Default IO)/Std. In (64 Bytes)/Input DWORD 11 @bit 16
//     Standard Inputs/MAIN.R4.In_From_HW/BYTE_[48] <-> Module 3 (Default IO)/Std. In (64 Bytes)/Input DWORD 11 @bit 24
//     Standard Inputs/MAIN.R4.In_From_HW/BYTE_[4] <-> Module 3 (Default IO)/Std. In (64 Bytes)/Input DWORD 0 @bit 24
//     Standard Inputs/MAIN.R4.In_From_HW/BYTE_[50] <-> Module 3 (Default IO)/Std. In (64 Bytes)/Input DWORD 12 @bit 8
//     Standard Inputs/MAIN.R4.In_From_HW/BYTE_[51] <-> Module 3 (Default IO)/Std. In (64 Bytes)/Input DWORD 12 @bit 16
//     Standard Inputs/MAIN.R4.In_From_HW/BYTE_[52] <-> Module 3 (Default IO)/Std. In (64 Bytes)/Input DWORD 12 @bit 24
//     Standard Inputs/MAIN.R4.In_From_HW/BYTE_[54] <-> Module 3 (Default IO)/Std. In (64 Bytes)/Input DWORD 13 @bit 8
//     Standard Inputs/MAIN.R4.In_From_HW/BYTE_[55] <-> Module 3 (Default IO)/Std. In (64 Bytes)/Input DWORD 13 @bit 16
//     Standard Inputs/MAIN.R4.In_From_HW/BYTE_[56] <-> Module 3 (Default IO)/Std. In (64 Bytes)/Input DWORD 13 @bit 24
//     Standard Inputs/MAIN.R4.In_From_HW/BYTE_[58] <-> Module 3 (Default IO)/Std. In (64 Bytes)/Input DWORD 14 @bit 8
//     Standard Inputs/MAIN.R4.In_From_HW/BYTE_[59] <-> Module 3 (Default IO)/Std. In (64 Bytes)/Input DWORD 14 @bit 16
//     Standard Inputs/MAIN.R4.In_From_HW/BYTE_[60] <-> Module 3 (Default IO)/Std. In (64 Bytes)/Input DWORD 14 @bit 24
//     Standard Inputs/MAIN.R4.In_From_HW/BYTE_[62] <-> Module 3 (Default IO)/Std. In (64 Bytes)/Input DWORD 15 @bit 8
//     Standard Inputs/MAIN.R4.In_From_HW/BYTE_[63] <-> Module 3 (Default IO)/Std. In (64 Bytes)/Input DWORD 15 @bit 16
//     Standard Inputs/MAIN.R4.In_From_HW/BYTE_[64] <-> Module 3 (Default IO)/Std. In (64 Bytes)/Input DWORD 15 @bit 24
//     Standard Inputs/MAIN.R4.In_From_HW/BYTE_[6] <-> Module 3 (Default IO)/Std. In (64 Bytes)/Input DWORD 1 @bit 8
//     Standard Inputs/MAIN.R4.In_From_HW/BYTE_[7] <-> Module 3 (Default IO)/Std. In (64 Bytes)/Input DWORD 1 @bit 16
//     Standard Inputs/MAIN.R4.In_From_HW/BYTE_[8] <-> Module 3 (Default IO)/Std. In (64 Bytes)/Input DWORD 1 @bit 24
//     Standard Inputs/MAIN.R4.In_From_HW/BYTE_[{1..61 step 4}] <-> Module 3 (Default IO)/Std. In (64 Bytes)/Input DWORD {0..15}  (16 links)
//     Standard Inputs/MAIN.R4.RT02/External_device_not_connected <-> Module 1 (Sync Inputs)/Compact/External device not connected
//     Standard Inputs/MAIN.R4.RT02/FSOE_Inputs_ConnID <-> Module 2 (Safety Data (8 Byte))/Inputs/FSOE/FSOE ConnID
//     Standard Inputs/MAIN.R4.RT02/FSOE_Inputs_Data_0 <-> Module 2 (Safety Data (8 Byte))/Inputs/FSOE/FSOE Data_0
//     Standard Inputs/MAIN.R4.RT02/FSOE_Inputs_Data_1 <-> Module 2 (Safety Data (8 Byte))/Inputs/FSOE/FSOE Data_1
//     Standard Inputs/MAIN.R4.RT02/FSOE_Inputs_Data_2 <-> Module 2 (Safety Data (8 Byte))/Inputs/FSOE/FSOE Data_2
//     Standard Inputs/MAIN.R4.RT02/FSOE_Inputs_Data_3 <-> Module 2 (Safety Data (8 Byte))/Inputs/FSOE/FSOE Data_3
//     Standard Inputs/MAIN.R4.RT02/InfoData/AdsAddr/netId <-> InfoData/AdsAddr/netId
//     Standard Inputs/MAIN.R4.RT02/InfoData/AdsAddr/port <-> InfoData/AdsAddr/port
//     Standard Inputs/MAIN.R4.RT02/InfoData/State <-> InfoData/State
//     Standard Inputs/MAIN.R4.RT02/TxPDO_State <-> Module 1 (Sync Inputs)/Compact/TxPDO state
//     Standard Inputs/MAIN.R4.RT02/TxPDO_Toogle <-> Module 1 (Sync Inputs)/Compact/TxPDO toggle
//     Standard Outputs/MAIN.R4.Out_To_HW/Byte_[10] <-> Module 3 (Default IO)/Std. Out (64 Bytes)/Output DWORD 2 @bit 8
//     Standard Outputs/MAIN.R4.Out_To_HW/Byte_[11] <-> Module 3 (Default IO)/Std. Out (64 Bytes)/Output DWORD 2 @bit 16
//     Standard Outputs/MAIN.R4.Out_To_HW/Byte_[12] <-> Module 3 (Default IO)/Std. Out (64 Bytes)/Output DWORD 2 @bit 24
//     Standard Outputs/MAIN.R4.Out_To_HW/Byte_[14] <-> Module 3 (Default IO)/Std. Out (64 Bytes)/Output DWORD 3 @bit 8
//     Standard Outputs/MAIN.R4.Out_To_HW/Byte_[15] <-> Module 3 (Default IO)/Std. Out (64 Bytes)/Output DWORD 3 @bit 16
//     Standard Outputs/MAIN.R4.Out_To_HW/Byte_[16] <-> Module 3 (Default IO)/Std. Out (64 Bytes)/Output DWORD 3 @bit 24
//     Standard Outputs/MAIN.R4.Out_To_HW/Byte_[18] <-> Module 3 (Default IO)/Std. Out (64 Bytes)/Output DWORD 4 @bit 8
//     Standard Outputs/MAIN.R4.Out_To_HW/Byte_[19] <-> Module 3 (Default IO)/Std. Out (64 Bytes)/Output DWORD 4 @bit 16
//     Standard Outputs/MAIN.R4.Out_To_HW/Byte_[20] <-> Module 3 (Default IO)/Std. Out (64 Bytes)/Output DWORD 4 @bit 24
//     Standard Outputs/MAIN.R4.Out_To_HW/Byte_[22] <-> Module 3 (Default IO)/Std. Out (64 Bytes)/Output DWORD 5 @bit 8
//     Standard Outputs/MAIN.R4.Out_To_HW/Byte_[23] <-> Module 3 (Default IO)/Std. Out (64 Bytes)/Output DWORD 5 @bit 16
//     Standard Outputs/MAIN.R4.Out_To_HW/Byte_[24] <-> Module 3 (Default IO)/Std. Out (64 Bytes)/Output DWORD 5 @bit 24
//     Standard Outputs/MAIN.R4.Out_To_HW/Byte_[26] <-> Module 3 (Default IO)/Std. Out (64 Bytes)/Output DWORD 6 @bit 8
//     Standard Outputs/MAIN.R4.Out_To_HW/Byte_[27] <-> Module 3 (Default IO)/Std. Out (64 Bytes)/Output DWORD 6 @bit 16
//     Standard Outputs/MAIN.R4.Out_To_HW/Byte_[28] <-> Module 3 (Default IO)/Std. Out (64 Bytes)/Output DWORD 6 @bit 24
//     Standard Outputs/MAIN.R4.Out_To_HW/Byte_[2] <-> Module 3 (Default IO)/Std. Out (64 Bytes)/Output DWORD 0 @bit 8
//     Standard Outputs/MAIN.R4.Out_To_HW/Byte_[30] <-> Module 3 (Default IO)/Std. Out (64 Bytes)/Output DWORD 7 @bit 8
//     Standard Outputs/MAIN.R4.Out_To_HW/Byte_[31] <-> Module 3 (Default IO)/Std. Out (64 Bytes)/Output DWORD 7 @bit 16
//     Standard Outputs/MAIN.R4.Out_To_HW/Byte_[32] <-> Module 3 (Default IO)/Std. Out (64 Bytes)/Output DWORD 7 @bit 24
//     Standard Outputs/MAIN.R4.Out_To_HW/Byte_[34] <-> Module 3 (Default IO)/Std. Out (64 Bytes)/Output DWORD 8 @bit 8
//     Standard Outputs/MAIN.R4.Out_To_HW/Byte_[35] <-> Module 3 (Default IO)/Std. Out (64 Bytes)/Output DWORD 8 @bit 16
//     Standard Outputs/MAIN.R4.Out_To_HW/Byte_[36] <-> Module 3 (Default IO)/Std. Out (64 Bytes)/Output DWORD 8 @bit 24
//     Standard Outputs/MAIN.R4.Out_To_HW/Byte_[38] <-> Module 3 (Default IO)/Std. Out (64 Bytes)/Output DWORD 9 @bit 8
//     Standard Outputs/MAIN.R4.Out_To_HW/Byte_[39] <-> Module 3 (Default IO)/Std. Out (64 Bytes)/Output DWORD 9 @bit 16
//     Standard Outputs/MAIN.R4.Out_To_HW/Byte_[3] <-> Module 3 (Default IO)/Std. Out (64 Bytes)/Output DWORD 0 @bit 16
//     Standard Outputs/MAIN.R4.Out_To_HW/Byte_[40] <-> Module 3 (Default IO)/Std. Out (64 Bytes)/Output DWORD 9 @bit 24
//     Standard Outputs/MAIN.R4.Out_To_HW/Byte_[42] <-> Module 3 (Default IO)/Std. Out (64 Bytes)/Output DWORD 10 @bit 8
//     Standard Outputs/MAIN.R4.Out_To_HW/Byte_[43] <-> Module 3 (Default IO)/Std. Out (64 Bytes)/Output DWORD 10 @bit 16
//     Standard Outputs/MAIN.R4.Out_To_HW/Byte_[44] <-> Module 3 (Default IO)/Std. Out (64 Bytes)/Output DWORD 10 @bit 24
//     Standard Outputs/MAIN.R4.Out_To_HW/Byte_[46] <-> Module 3 (Default IO)/Std. Out (64 Bytes)/Output DWORD 11 @bit 8
//     Standard Outputs/MAIN.R4.Out_To_HW/Byte_[47] <-> Module 3 (Default IO)/Std. Out (64 Bytes)/Output DWORD 11 @bit 16
//     Standard Outputs/MAIN.R4.Out_To_HW/Byte_[48] <-> Module 3 (Default IO)/Std. Out (64 Bytes)/Output DWORD 11 @bit 24
//     Standard Outputs/MAIN.R4.Out_To_HW/Byte_[4] <-> Module 3 (Default IO)/Std. Out (64 Bytes)/Output DWORD 0 @bit 24
//     Standard Outputs/MAIN.R4.Out_To_HW/Byte_[50] <-> Module 3 (Default IO)/Std. Out (64 Bytes)/Output DWORD 12 @bit 8
//     Standard Outputs/MAIN.R4.Out_To_HW/Byte_[51] <-> Module 3 (Default IO)/Std. Out (64 Bytes)/Output DWORD 12 @bit 16
//     Standard Outputs/MAIN.R4.Out_To_HW/Byte_[52] <-> Module 3 (Default IO)/Std. Out (64 Bytes)/Output DWORD 12 @bit 24
//     Standard Outputs/MAIN.R4.Out_To_HW/Byte_[54] <-> Module 3 (Default IO)/Std. Out (64 Bytes)/Output DWORD 13 @bit 8
//     Standard Outputs/MAIN.R4.Out_To_HW/Byte_[55] <-> Module 3 (Default IO)/Std. Out (64 Bytes)/Output DWORD 13 @bit 16
//     Standard Outputs/MAIN.R4.Out_To_HW/Byte_[56] <-> Module 3 (Default IO)/Std. Out (64 Bytes)/Output DWORD 13 @bit 24
//     Standard Outputs/MAIN.R4.Out_To_HW/Byte_[58] <-> Module 3 (Default IO)/Std. Out (64 Bytes)/Output DWORD 14 @bit 8
//     Standard Outputs/MAIN.R4.Out_To_HW/Byte_[59] <-> Module 3 (Default IO)/Std. Out (64 Bytes)/Output DWORD 14 @bit 16
//     Standard Outputs/MAIN.R4.Out_To_HW/Byte_[60] <-> Module 3 (Default IO)/Std. Out (64 Bytes)/Output DWORD 14 @bit 24
//     Standard Outputs/MAIN.R4.Out_To_HW/Byte_[62] <-> Module 3 (Default IO)/Std. Out (64 Bytes)/Output DWORD 15 @bit 8
//     Standard Outputs/MAIN.R4.Out_To_HW/Byte_[63] <-> Module 3 (Default IO)/Std. Out (64 Bytes)/Output DWORD 15 @bit 16
//     Standard Outputs/MAIN.R4.Out_To_HW/Byte_[64] <-> Module 3 (Default IO)/Std. Out (64 Bytes)/Output DWORD 15 @bit 24
//     Standard Outputs/MAIN.R4.Out_To_HW/Byte_[6] <-> Module 3 (Default IO)/Std. Out (64 Bytes)/Output DWORD 1 @bit 8
//     Standard Outputs/MAIN.R4.Out_To_HW/Byte_[7] <-> Module 3 (Default IO)/Std. Out (64 Bytes)/Output DWORD 1 @bit 16
//     Standard Outputs/MAIN.R4.Out_To_HW/Byte_[8] <-> Module 3 (Default IO)/Std. Out (64 Bytes)/Output DWORD 1 @bit 24
//     Standard Outputs/MAIN.R4.Out_To_HW/Byte_[{1..61 step 4}] <-> Module 3 (Default IO)/Std. Out (64 Bytes)/Output DWORD {0..15}  (16 links)
//   SODG11_SSCC610_2403701_PLC/SODG11_SSCC610_2403701_PLC Instance <-> EtherCAT Master (EtherCAT)/R4.T01 (EK1100)
//     Standard Inputs/MAIN.R4.T01/InfoData/State <-> InfoData/State
//   SODG11_SSCC610_2403701_PLC/SODG11_SSCC610_2403701_PLC Instance <-> EtherCAT Master (EtherCAT)/R4.T01 (EK1100)/R4.T02 (EL6900)
//     Standard Inputs/MAIN.R4.RT02/FSOE_Outputs_Data_0 @bit 1 <-> StandardInputs/Standard Out Var 14
//     Standard Inputs/MAIN.R4.RT02/FSOE_Outputs_Data_0 @bit 2 <-> StandardInputs/Standard Out Var 15
//     Standard Inputs/MAIN.R4.RT02/FSOE_Outputs_Data_2 @bit 1 <-> StandardInputs/Standard Out Var 18
//     Standard Inputs/MAIN.R4.RT02/FSOE_Outputs_Data_2 <-> StandardInputs/Standard Out Var 17
//     Standard Inputs/MAIN.R4.T02_STAT/Device_Info_Data/Project_CRC <-> Device Info Data/Project CRC
//     Standard Inputs/MAIN.R4.T02_STAT/FBs_FB_ERR <-> StandardInputs/Standard Out Var 16
//     Standard Inputs/MAIN.R4.T02_STAT/FBs_FB_ERR @bit 16 <-> StandardInputs/Standard Out Var 19
//     Standard Inputs/MAIN.R4.T02_STAT/FBs_FB_ERR @bit 29 <-> StandardInputs/Standard Out Var 20
//     Standard Inputs/MAIN.R4.T02_STAT/InfoData/AdsAddr/netId <-> InfoData/AdsAddr/netId
//     Standard Inputs/MAIN.R4.T02_STAT/InfoData/AdsAddr/port <-> InfoData/AdsAddr/port
//     Standard Inputs/MAIN.R4.T02_STAT/InfoData/State <-> InfoData/State
//     Standard Inputs/MAIN.R4.T02_STAT/SGs_COM_ERR @bit 1 <-> StandardInputs/Standard Out Var 12
//     Standard Inputs/MAIN.R4.T02_STAT/SGs_COM_ERR <-> StandardInputs/Standard Out Var 9
//     Standard Inputs/MAIN.R4.T02_STAT/SGs_FB_ERR @bit 1 <-> StandardInputs/Standard Out Var 11
//     Standard Inputs/MAIN.R4.T02_STAT/SGs_FB_ERR <-> StandardInputs/Standard Out Var 8
//     Standard Inputs/MAIN.R4.T02_STAT/SGs_OUT_ERR <-> StandardInputs/Standard Out Var 10
//     Standard Inputs/MAIN.R4.T02_STAT/SGs_OUT_ERR @bit 1 <-> StandardInputs/Standard Out Var 13
//     Standard Outputs/MAIN.R4.T02_CMD/FBs_ControlPowerPB <-> StandardOutputs/Standard In Var 7
//     Standard Outputs/MAIN.R4.T02_CMD/SGs_ERRAck <-> StandardOutputs/Standard In Var 4
//     Standard Outputs/MAIN.R4.T02_CMD/SGs_ERRAck <-> StandardOutputs/Standard In Var 6
//     Standard Outputs/MAIN.R4.T02_CMD/SGs_RUNSTOP <-> StandardOutputs/Standard In Var 3
//     Standard Outputs/MAIN.R4.T02_CMD/SGs_RUNSTOP <-> StandardOutputs/Standard In Var 5
//     Standard Outputs/MAIN.Safety_Zone_Test <-> StandardOutputs/Standard In Var 21
//   SODG11_SSCC610_2403701_PLC/SODG11_SSCC610_2403701_PLC Instance <-> EtherCAT Master (EtherCAT)/R4.T01 (EK1100)/R4.T03 (EL1904)
//     Standard Inputs/MAIN.R4.T03/I <-> Module 1 (FSOES)/TxPDO/FSOE/InputChannel1
//     Standard Inputs/MAIN.R4.T03/I @bit 1 <-> Module 1 (FSOES)/TxPDO/FSOE/InputChannel2
//     Standard Inputs/MAIN.R4.T03/I @bit 2 <-> Module 1 (FSOES)/TxPDO/FSOE/InputChannel3
//     Standard Inputs/MAIN.R4.T03/I @bit 3 <-> Module 1 (FSOES)/TxPDO/FSOE/InputChannel4
//     Standard Inputs/MAIN.R4.T03/InfoData/State <-> InfoData/State
//   SODG11_SSCC610_2403701_PLC/SODG11_SSCC610_2403701_PLC Instance <-> EtherCAT Master (EtherCAT)/R4.T01 (EK1100)/R4.T04 (EK1122)
//     Standard Inputs/MAIN.R4.T04/InfoData/State <-> InfoData/State
//   SODG11_SSCC610_2403701_PLC/SODG11_SSCC610_2403701_PLC Instance <-> EtherCAT Master (EtherCAT)/R4.T01 (EK1100)/R4.T04 (EK1122)/EOAT04.N01 (EP1008-0002)
//     Standard Inputs/EOAT04.N01/I <-> Channel 1/Input
//     Standard Inputs/EOAT04.N01/I @bit 1 <-> Channel 2/Input
//     Standard Inputs/EOAT04.N01/I @bit 2 <-> Channel 3/Input
//     Standard Inputs/EOAT04.N01/I @bit 3 <-> Channel 4/Input
//     Standard Inputs/EOAT04.N01/I @bit 4 <-> Channel 5/Input
//     Standard Inputs/EOAT04.N01/I @bit 5 <-> Channel 6/Input
//     Standard Inputs/EOAT04.N01/I @bit 6 <-> Channel 7/Input
//     Standard Inputs/EOAT04.N01/I @bit 7 <-> Channel 8/Input
//     Standard Inputs/EOAT04.N01/InfoData/State <-> InfoData/State
//     Standard Inputs/EOAT04.N01/Wc_State <-> WcState/WcState
//   SODG11_SSCC610_2403701_PLC/SODG11_SSCC610_2403701_PLC Instance <-> EtherCAT Master (EtherCAT)/R4.T01 (EK1100)/R4.T04 (EK1122)/EOAT04.N02 (EP1008-0002)
//     Standard Inputs/EOAT04.N02/I <-> Channel 1/Input
//     Standard Inputs/EOAT04.N02/I @bit 1 <-> Channel 2/Input
//     Standard Inputs/EOAT04.N02/I @bit 2 <-> Channel 3/Input
//     Standard Inputs/EOAT04.N02/I @bit 3 <-> Channel 4/Input
//     Standard Inputs/EOAT04.N02/I @bit 4 <-> Channel 5/Input
//     Standard Inputs/EOAT04.N02/I @bit 5 <-> Channel 6/Input
//     Standard Inputs/EOAT04.N02/I @bit 6 <-> Channel 7/Input
//     Standard Inputs/EOAT04.N02/I @bit 7 <-> Channel 8/Input
//     Standard Inputs/EOAT04.N02/InfoData/State <-> InfoData/State
//     Standard Inputs/EOAT04.N02/Wc_State <-> WcState/WcState
//   SODG11_SSCC610_2403701_PLC/SODG11_SSCC610_2403701_PLC Instance <-> EtherCAT Master (EtherCAT)/R4.T01 (EK1100)/R4.T04 (EK1122)/EOAT04.N03 (EP1008-0002)
//     Standard Inputs/EOAT04.N03/I <-> Channel 1/Input
//     Standard Inputs/EOAT04.N03/I @bit 1 <-> Channel 2/Input
//     Standard Inputs/EOAT04.N03/I @bit 2 <-> Channel 3/Input
//     Standard Inputs/EOAT04.N03/I @bit 3 <-> Channel 4/Input
//     Standard Inputs/EOAT04.N03/I @bit 4 <-> Channel 5/Input
//     Standard Inputs/EOAT04.N03/I @bit 5 <-> Channel 6/Input
//     Standard Inputs/EOAT04.N03/I @bit 6 <-> Channel 7/Input
//     Standard Inputs/EOAT04.N03/I @bit 7 <-> Channel 8/Input
//     Standard Inputs/EOAT04.N03/InfoData/State <-> InfoData/State
//     Standard Inputs/EOAT04.N03/Wc_State <-> WcState/WcState
//   SODG11_SSCC610_2403701_PLC/SODG11_SSCC610_2403701_PLC Instance <-> EtherCAT Master (EtherCAT)/R4.T01 (EK1100)/R4.T04 (EK1122)/EOAT04.N04 (EP1008-0002)
//     Standard Inputs/EOAT04.N04/I <-> Channel 1/Input
//     Standard Inputs/EOAT04.N04/I @bit 1 <-> Channel 2/Input
//     Standard Inputs/EOAT04.N04/I @bit 2 <-> Channel 3/Input
//     Standard Inputs/EOAT04.N04/I @bit 3 <-> Channel 4/Input
//     Standard Inputs/EOAT04.N04/I @bit 4 <-> Channel 5/Input
//     Standard Inputs/EOAT04.N04/I @bit 5 <-> Channel 6/Input
//     Standard Inputs/EOAT04.N04/I @bit 6 <-> Channel 7/Input
//     Standard Inputs/EOAT04.N04/I @bit 7 <-> Channel 8/Input
//     Standard Inputs/EOAT04.N04/InfoData/State <-> InfoData/State
//     Standard Inputs/EOAT04.N04/Wc_State <-> WcState/WcState
//   SODG11_SSCC610_2403701_PLC/SODG11_SSCC610_2403701_PLC Instance <-> EtherCAT Master (EtherCAT)/R4.T01 (EK1100)/R4.T04 (EK1122)/EOAT04.N100 (EX260-SEC1)
//     Standard Inputs/EOAT04.N100_STAT/InfoData/State <-> InfoData/State
//     Standard Outputs/EOAT04.N100/Q <-> Byte 0/Output
//     Standard Outputs/EOAT04.N100/Q @bit 8 <-> Byte 1/Output
//     Standard Outputs/EOAT04.N100/Q @bit 16 <-> Byte 2/Output
//     Standard Outputs/EOAT04.N100/Q @bit 24 <-> Byte 3/Output
//   SODG11_SSCC610_2403701_PLC/SODG11_SSCC610_2403701_PLC Instance <-> EtherCAT Master (EtherCAT)/R5.RT02 (EL6695-1001)
//     Standard Inputs/MAIN.R5.In_From_HW/BYTE_[10] <-> Module 3 (Default IO)/Std. In (64 Bytes)/Input DWORD 2 @bit 8
//     Standard Inputs/MAIN.R5.In_From_HW/BYTE_[11] <-> Module 3 (Default IO)/Std. In (64 Bytes)/Input DWORD 2 @bit 16
//     Standard Inputs/MAIN.R5.In_From_HW/BYTE_[12] <-> Module 3 (Default IO)/Std. In (64 Bytes)/Input DWORD 2 @bit 24
//     Standard Inputs/MAIN.R5.In_From_HW/BYTE_[14] <-> Module 3 (Default IO)/Std. In (64 Bytes)/Input DWORD 3 @bit 8
//     Standard Inputs/MAIN.R5.In_From_HW/BYTE_[15] <-> Module 3 (Default IO)/Std. In (64 Bytes)/Input DWORD 3 @bit 16
//     Standard Inputs/MAIN.R5.In_From_HW/BYTE_[16] <-> Module 3 (Default IO)/Std. In (64 Bytes)/Input DWORD 3 @bit 24
//     Standard Inputs/MAIN.R5.In_From_HW/BYTE_[18] <-> Module 3 (Default IO)/Std. In (64 Bytes)/Input DWORD 4 @bit 8
//     Standard Inputs/MAIN.R5.In_From_HW/BYTE_[19] <-> Module 3 (Default IO)/Std. In (64 Bytes)/Input DWORD 4 @bit 16
//     Standard Inputs/MAIN.R5.In_From_HW/BYTE_[20] <-> Module 3 (Default IO)/Std. In (64 Bytes)/Input DWORD 4 @bit 24
//     Standard Inputs/MAIN.R5.In_From_HW/BYTE_[22] <-> Module 3 (Default IO)/Std. In (64 Bytes)/Input DWORD 5 @bit 8
//     Standard Inputs/MAIN.R5.In_From_HW/BYTE_[23] <-> Module 3 (Default IO)/Std. In (64 Bytes)/Input DWORD 5 @bit 16
//     Standard Inputs/MAIN.R5.In_From_HW/BYTE_[24] <-> Module 3 (Default IO)/Std. In (64 Bytes)/Input DWORD 5 @bit 24
//     Standard Inputs/MAIN.R5.In_From_HW/BYTE_[26] <-> Module 3 (Default IO)/Std. In (64 Bytes)/Input DWORD 6 @bit 8
//     Standard Inputs/MAIN.R5.In_From_HW/BYTE_[27] <-> Module 3 (Default IO)/Std. In (64 Bytes)/Input DWORD 6 @bit 16
//     Standard Inputs/MAIN.R5.In_From_HW/BYTE_[28] <-> Module 3 (Default IO)/Std. In (64 Bytes)/Input DWORD 6 @bit 24
//     Standard Inputs/MAIN.R5.In_From_HW/BYTE_[2] <-> Module 3 (Default IO)/Std. In (64 Bytes)/Input DWORD 0 @bit 8
//     Standard Inputs/MAIN.R5.In_From_HW/BYTE_[30] <-> Module 3 (Default IO)/Std. In (64 Bytes)/Input DWORD 7 @bit 8
//     Standard Inputs/MAIN.R5.In_From_HW/BYTE_[31] <-> Module 3 (Default IO)/Std. In (64 Bytes)/Input DWORD 7 @bit 16
//     Standard Inputs/MAIN.R5.In_From_HW/BYTE_[32] <-> Module 3 (Default IO)/Std. In (64 Bytes)/Input DWORD 7 @bit 24
//     Standard Inputs/MAIN.R5.In_From_HW/BYTE_[34] <-> Module 3 (Default IO)/Std. In (64 Bytes)/Input DWORD 8 @bit 8
//     Standard Inputs/MAIN.R5.In_From_HW/BYTE_[35] <-> Module 3 (Default IO)/Std. In (64 Bytes)/Input DWORD 8 @bit 16
//     Standard Inputs/MAIN.R5.In_From_HW/BYTE_[36] <-> Module 3 (Default IO)/Std. In (64 Bytes)/Input DWORD 8 @bit 24
//     Standard Inputs/MAIN.R5.In_From_HW/BYTE_[38] <-> Module 3 (Default IO)/Std. In (64 Bytes)/Input DWORD 9 @bit 8
//     Standard Inputs/MAIN.R5.In_From_HW/BYTE_[39] <-> Module 3 (Default IO)/Std. In (64 Bytes)/Input DWORD 9 @bit 16
//     Standard Inputs/MAIN.R5.In_From_HW/BYTE_[3] <-> Module 3 (Default IO)/Std. In (64 Bytes)/Input DWORD 0 @bit 16
//     Standard Inputs/MAIN.R5.In_From_HW/BYTE_[40] <-> Module 3 (Default IO)/Std. In (64 Bytes)/Input DWORD 9 @bit 24
//     Standard Inputs/MAIN.R5.In_From_HW/BYTE_[42] <-> Module 3 (Default IO)/Std. In (64 Bytes)/Input DWORD 10 @bit 8
//     Standard Inputs/MAIN.R5.In_From_HW/BYTE_[43] <-> Module 3 (Default IO)/Std. In (64 Bytes)/Input DWORD 10 @bit 16
//     Standard Inputs/MAIN.R5.In_From_HW/BYTE_[44] <-> Module 3 (Default IO)/Std. In (64 Bytes)/Input DWORD 10 @bit 24
//     Standard Inputs/MAIN.R5.In_From_HW/BYTE_[46] <-> Module 3 (Default IO)/Std. In (64 Bytes)/Input DWORD 11 @bit 8
//     Standard Inputs/MAIN.R5.In_From_HW/BYTE_[47] <-> Module 3 (Default IO)/Std. In (64 Bytes)/Input DWORD 11 @bit 16
//     Standard Inputs/MAIN.R5.In_From_HW/BYTE_[48] <-> Module 3 (Default IO)/Std. In (64 Bytes)/Input DWORD 11 @bit 24
//     Standard Inputs/MAIN.R5.In_From_HW/BYTE_[4] <-> Module 3 (Default IO)/Std. In (64 Bytes)/Input DWORD 0 @bit 24
//     Standard Inputs/MAIN.R5.In_From_HW/BYTE_[50] <-> Module 3 (Default IO)/Std. In (64 Bytes)/Input DWORD 12 @bit 8
//     Standard Inputs/MAIN.R5.In_From_HW/BYTE_[51] <-> Module 3 (Default IO)/Std. In (64 Bytes)/Input DWORD 12 @bit 16
//     Standard Inputs/MAIN.R5.In_From_HW/BYTE_[52] <-> Module 3 (Default IO)/Std. In (64 Bytes)/Input DWORD 12 @bit 24
//     Standard Inputs/MAIN.R5.In_From_HW/BYTE_[54] <-> Module 3 (Default IO)/Std. In (64 Bytes)/Input DWORD 13 @bit 8
//     Standard Inputs/MAIN.R5.In_From_HW/BYTE_[55] <-> Module 3 (Default IO)/Std. In (64 Bytes)/Input DWORD 13 @bit 16
//     Standard Inputs/MAIN.R5.In_From_HW/BYTE_[56] <-> Module 3 (Default IO)/Std. In (64 Bytes)/Input DWORD 13 @bit 24
//     Standard Inputs/MAIN.R5.In_From_HW/BYTE_[58] <-> Module 3 (Default IO)/Std. In (64 Bytes)/Input DWORD 14 @bit 8
//     Standard Inputs/MAIN.R5.In_From_HW/BYTE_[59] <-> Module 3 (Default IO)/Std. In (64 Bytes)/Input DWORD 14 @bit 16
//     Standard Inputs/MAIN.R5.In_From_HW/BYTE_[60] <-> Module 3 (Default IO)/Std. In (64 Bytes)/Input DWORD 14 @bit 24
//     Standard Inputs/MAIN.R5.In_From_HW/BYTE_[62] <-> Module 3 (Default IO)/Std. In (64 Bytes)/Input DWORD 15 @bit 8
//     Standard Inputs/MAIN.R5.In_From_HW/BYTE_[63] <-> Module 3 (Default IO)/Std. In (64 Bytes)/Input DWORD 15 @bit 16
//     Standard Inputs/MAIN.R5.In_From_HW/BYTE_[64] <-> Module 3 (Default IO)/Std. In (64 Bytes)/Input DWORD 15 @bit 24
//     Standard Inputs/MAIN.R5.In_From_HW/BYTE_[6] <-> Module 3 (Default IO)/Std. In (64 Bytes)/Input DWORD 1 @bit 8
//     Standard Inputs/MAIN.R5.In_From_HW/BYTE_[7] <-> Module 3 (Default IO)/Std. In (64 Bytes)/Input DWORD 1 @bit 16
//     Standard Inputs/MAIN.R5.In_From_HW/BYTE_[8] <-> Module 3 (Default IO)/Std. In (64 Bytes)/Input DWORD 1 @bit 24
//     Standard Inputs/MAIN.R5.In_From_HW/BYTE_[{1..61 step 4}] <-> Module 3 (Default IO)/Std. In (64 Bytes)/Input DWORD {0..15}  (16 links)
//     Standard Inputs/MAIN.R5.RT02/External_device_not_connected <-> Module 1 (Sync Inputs)/Compact/External device not connected
//     Standard Inputs/MAIN.R5.RT02/FSOE_Inputs_ConnID <-> Module 2 (Safety Data (8 Byte))/Inputs/FSOE/FSOE ConnID
//     Standard Inputs/MAIN.R5.RT02/FSOE_Inputs_Data_0 <-> Module 2 (Safety Data (8 Byte))/Inputs/FSOE/FSOE Data_0
//     Standard Inputs/MAIN.R5.RT02/FSOE_Inputs_Data_1 <-> Module 2 (Safety Data (8 Byte))/Inputs/FSOE/FSOE Data_1
//     Standard Inputs/MAIN.R5.RT02/FSOE_Inputs_Data_2 <-> Module 2 (Safety Data (8 Byte))/Inputs/FSOE/FSOE Data_2
//     Standard Inputs/MAIN.R5.RT02/FSOE_Inputs_Data_3 <-> Module 2 (Safety Data (8 Byte))/Inputs/FSOE/FSOE Data_3
//     Standard Inputs/MAIN.R5.RT02/InfoData/AdsAddr/netId <-> InfoData/AdsAddr/netId
//     Standard Inputs/MAIN.R5.RT02/InfoData/AdsAddr/port <-> InfoData/AdsAddr/port
//     Standard Inputs/MAIN.R5.RT02/InfoData/State <-> InfoData/State
//     Standard Inputs/MAIN.R5.RT02/TxPDO_State <-> Module 1 (Sync Inputs)/Compact/TxPDO state
//     Standard Inputs/MAIN.R5.RT02/TxPDO_Toogle <-> Module 1 (Sync Inputs)/Compact/TxPDO toggle
//     Standard Outputs/MAIN.R5.Out_To_HW/Byte_[10] <-> Module 3 (Default IO)/Std. Out (64 Bytes)/Output DWORD 2 @bit 8
//     Standard Outputs/MAIN.R5.Out_To_HW/Byte_[11] <-> Module 3 (Default IO)/Std. Out (64 Bytes)/Output DWORD 2 @bit 16
//     Standard Outputs/MAIN.R5.Out_To_HW/Byte_[12] <-> Module 3 (Default IO)/Std. Out (64 Bytes)/Output DWORD 2 @bit 24
//     Standard Outputs/MAIN.R5.Out_To_HW/Byte_[14] <-> Module 3 (Default IO)/Std. Out (64 Bytes)/Output DWORD 3 @bit 8
//     Standard Outputs/MAIN.R5.Out_To_HW/Byte_[15] <-> Module 3 (Default IO)/Std. Out (64 Bytes)/Output DWORD 3 @bit 16
//     Standard Outputs/MAIN.R5.Out_To_HW/Byte_[16] <-> Module 3 (Default IO)/Std. Out (64 Bytes)/Output DWORD 3 @bit 24
//     Standard Outputs/MAIN.R5.Out_To_HW/Byte_[18] <-> Module 3 (Default IO)/Std. Out (64 Bytes)/Output DWORD 4 @bit 8
//     Standard Outputs/MAIN.R5.Out_To_HW/Byte_[19] <-> Module 3 (Default IO)/Std. Out (64 Bytes)/Output DWORD 4 @bit 16
//     Standard Outputs/MAIN.R5.Out_To_HW/Byte_[20] <-> Module 3 (Default IO)/Std. Out (64 Bytes)/Output DWORD 4 @bit 24
//     Standard Outputs/MAIN.R5.Out_To_HW/Byte_[22] <-> Module 3 (Default IO)/Std. Out (64 Bytes)/Output DWORD 5 @bit 8
//     Standard Outputs/MAIN.R5.Out_To_HW/Byte_[23] <-> Module 3 (Default IO)/Std. Out (64 Bytes)/Output DWORD 5 @bit 16
//     Standard Outputs/MAIN.R5.Out_To_HW/Byte_[24] <-> Module 3 (Default IO)/Std. Out (64 Bytes)/Output DWORD 5 @bit 24
//     Standard Outputs/MAIN.R5.Out_To_HW/Byte_[26] <-> Module 3 (Default IO)/Std. Out (64 Bytes)/Output DWORD 6 @bit 8
//     Standard Outputs/MAIN.R5.Out_To_HW/Byte_[27] <-> Module 3 (Default IO)/Std. Out (64 Bytes)/Output DWORD 6 @bit 16
//     Standard Outputs/MAIN.R5.Out_To_HW/Byte_[28] <-> Module 3 (Default IO)/Std. Out (64 Bytes)/Output DWORD 6 @bit 24
//     Standard Outputs/MAIN.R5.Out_To_HW/Byte_[2] <-> Module 3 (Default IO)/Std. Out (64 Bytes)/Output DWORD 0 @bit 8
//     Standard Outputs/MAIN.R5.Out_To_HW/Byte_[30] <-> Module 3 (Default IO)/Std. Out (64 Bytes)/Output DWORD 7 @bit 8
//     Standard Outputs/MAIN.R5.Out_To_HW/Byte_[31] <-> Module 3 (Default IO)/Std. Out (64 Bytes)/Output DWORD 7 @bit 16
//     Standard Outputs/MAIN.R5.Out_To_HW/Byte_[32] <-> Module 3 (Default IO)/Std. Out (64 Bytes)/Output DWORD 7 @bit 24
//     Standard Outputs/MAIN.R5.Out_To_HW/Byte_[34] <-> Module 3 (Default IO)/Std. Out (64 Bytes)/Output DWORD 8 @bit 8
//     Standard Outputs/MAIN.R5.Out_To_HW/Byte_[35] <-> Module 3 (Default IO)/Std. Out (64 Bytes)/Output DWORD 8 @bit 16
//     Standard Outputs/MAIN.R5.Out_To_HW/Byte_[36] <-> Module 3 (Default IO)/Std. Out (64 Bytes)/Output DWORD 8 @bit 24
//     Standard Outputs/MAIN.R5.Out_To_HW/Byte_[38] <-> Module 3 (Default IO)/Std. Out (64 Bytes)/Output DWORD 9 @bit 8
//     Standard Outputs/MAIN.R5.Out_To_HW/Byte_[39] <-> Module 3 (Default IO)/Std. Out (64 Bytes)/Output DWORD 9 @bit 16
//     Standard Outputs/MAIN.R5.Out_To_HW/Byte_[3] <-> Module 3 (Default IO)/Std. Out (64 Bytes)/Output DWORD 0 @bit 16
//     Standard Outputs/MAIN.R5.Out_To_HW/Byte_[40] <-> Module 3 (Default IO)/Std. Out (64 Bytes)/Output DWORD 9 @bit 24
//     Standard Outputs/MAIN.R5.Out_To_HW/Byte_[42] <-> Module 3 (Default IO)/Std. Out (64 Bytes)/Output DWORD 10 @bit 8
//     Standard Outputs/MAIN.R5.Out_To_HW/Byte_[43] <-> Module 3 (Default IO)/Std. Out (64 Bytes)/Output DWORD 10 @bit 16
//     Standard Outputs/MAIN.R5.Out_To_HW/Byte_[44] <-> Module 3 (Default IO)/Std. Out (64 Bytes)/Output DWORD 10 @bit 24
//     Standard Outputs/MAIN.R5.Out_To_HW/Byte_[46] <-> Module 3 (Default IO)/Std. Out (64 Bytes)/Output DWORD 11 @bit 8
//     Standard Outputs/MAIN.R5.Out_To_HW/Byte_[47] <-> Module 3 (Default IO)/Std. Out (64 Bytes)/Output DWORD 11 @bit 16
//     Standard Outputs/MAIN.R5.Out_To_HW/Byte_[48] <-> Module 3 (Default IO)/Std. Out (64 Bytes)/Output DWORD 11 @bit 24
//     Standard Outputs/MAIN.R5.Out_To_HW/Byte_[4] <-> Module 3 (Default IO)/Std. Out (64 Bytes)/Output DWORD 0 @bit 24
//     Standard Outputs/MAIN.R5.Out_To_HW/Byte_[50] <-> Module 3 (Default IO)/Std. Out (64 Bytes)/Output DWORD 12 @bit 8
//     Standard Outputs/MAIN.R5.Out_To_HW/Byte_[51] <-> Module 3 (Default IO)/Std. Out (64 Bytes)/Output DWORD 12 @bit 16
//     Standard Outputs/MAIN.R5.Out_To_HW/Byte_[52] <-> Module 3 (Default IO)/Std. Out (64 Bytes)/Output DWORD 12 @bit 24
//     Standard Outputs/MAIN.R5.Out_To_HW/Byte_[54] <-> Module 3 (Default IO)/Std. Out (64 Bytes)/Output DWORD 13 @bit 8
//     Standard Outputs/MAIN.R5.Out_To_HW/Byte_[55] <-> Module 3 (Default IO)/Std. Out (64 Bytes)/Output DWORD 13 @bit 16
//     Standard Outputs/MAIN.R5.Out_To_HW/Byte_[56] <-> Module 3 (Default IO)/Std. Out (64 Bytes)/Output DWORD 13 @bit 24
//     Standard Outputs/MAIN.R5.Out_To_HW/Byte_[58] <-> Module 3 (Default IO)/Std. Out (64 Bytes)/Output DWORD 14 @bit 8
//     Standard Outputs/MAIN.R5.Out_To_HW/Byte_[59] <-> Module 3 (Default IO)/Std. Out (64 Bytes)/Output DWORD 14 @bit 16
//     Standard Outputs/MAIN.R5.Out_To_HW/Byte_[60] <-> Module 3 (Default IO)/Std. Out (64 Bytes)/Output DWORD 14 @bit 24
//     Standard Outputs/MAIN.R5.Out_To_HW/Byte_[62] <-> Module 3 (Default IO)/Std. Out (64 Bytes)/Output DWORD 15 @bit 8
//     Standard Outputs/MAIN.R5.Out_To_HW/Byte_[63] <-> Module 3 (Default IO)/Std. Out (64 Bytes)/Output DWORD 15 @bit 16
//     Standard Outputs/MAIN.R5.Out_To_HW/Byte_[64] <-> Module 3 (Default IO)/Std. Out (64 Bytes)/Output DWORD 15 @bit 24
//     Standard Outputs/MAIN.R5.Out_To_HW/Byte_[6] <-> Module 3 (Default IO)/Std. Out (64 Bytes)/Output DWORD 1 @bit 8
//     Standard Outputs/MAIN.R5.Out_To_HW/Byte_[7] <-> Module 3 (Default IO)/Std. Out (64 Bytes)/Output DWORD 1 @bit 16
//     Standard Outputs/MAIN.R5.Out_To_HW/Byte_[8] <-> Module 3 (Default IO)/Std. Out (64 Bytes)/Output DWORD 1 @bit 24
//     Standard Outputs/MAIN.R5.Out_To_HW/Byte_[{1..61 step 4}] <-> Module 3 (Default IO)/Std. Out (64 Bytes)/Output DWORD {0..15}  (16 links)
//   SODG11_SSCC610_2403701_PLC/SODG11_SSCC610_2403701_PLC Instance <-> EtherCAT Master (EtherCAT)/R5.T01 (EK1100)
//     Standard Inputs/MAIN.R5.T01/InfoData/State <-> InfoData/State
//   SODG11_SSCC610_2403701_PLC/SODG11_SSCC610_2403701_PLC Instance <-> EtherCAT Master (EtherCAT)/R5.T01 (EK1100)/R5.T02 (EL6900)
//     Standard Inputs/MAIN.R5.RT02/FSOE_Outputs_Data_0 @bit 1 <-> StandardInputs/Standard Out Var 14
//     Standard Inputs/MAIN.R5.RT02/FSOE_Outputs_Data_0 @bit 2 <-> StandardInputs/Standard Out Var 15
//     Standard Inputs/MAIN.R5.RT02/FSOE_Outputs_Data_2 @bit 1 <-> StandardInputs/Standard Out Var 18
//     Standard Inputs/MAIN.R5.RT02/FSOE_Outputs_Data_2 <-> StandardInputs/Standard Out Var 17
//     Standard Inputs/MAIN.R5.T02_STAT/Device_Info_Data/Project_CRC <-> Device Info Data/Project CRC
//     Standard Inputs/MAIN.R5.T02_STAT/FBs_FB_ERR <-> StandardInputs/Standard Out Var 16
//     Standard Inputs/MAIN.R5.T02_STAT/FBs_FB_ERR @bit 16 <-> StandardInputs/Standard Out Var 19
//     Standard Inputs/MAIN.R5.T02_STAT/FBs_FB_ERR @bit 29 <-> StandardInputs/Standard Out Var 20
//     Standard Inputs/MAIN.R5.T02_STAT/InfoData/AdsAddr/netId <-> InfoData/AdsAddr/netId
//     Standard Inputs/MAIN.R5.T02_STAT/InfoData/AdsAddr/port <-> InfoData/AdsAddr/port
//     Standard Inputs/MAIN.R5.T02_STAT/InfoData/State <-> InfoData/State
//     Standard Inputs/MAIN.R5.T02_STAT/SGs_COM_ERR @bit 1 <-> StandardInputs/Standard Out Var 12
//     Standard Inputs/MAIN.R5.T02_STAT/SGs_COM_ERR <-> StandardInputs/Standard Out Var 9
//     Standard Inputs/MAIN.R5.T02_STAT/SGs_FB_ERR @bit 1 <-> StandardInputs/Standard Out Var 11
//     Standard Inputs/MAIN.R5.T02_STAT/SGs_FB_ERR <-> StandardInputs/Standard Out Var 8
//     Standard Inputs/MAIN.R5.T02_STAT/SGs_OUT_ERR <-> StandardInputs/Standard Out Var 10
//     Standard Inputs/MAIN.R5.T02_STAT/SGs_OUT_ERR @bit 1 <-> StandardInputs/Standard Out Var 13
//     Standard Outputs/MAIN.R5.T02_CMD/FBs_ControlPowerPB <-> StandardOutputs/Standard In Var 7
//     Standard Outputs/MAIN.R5.T02_CMD/SGs_ERRAck <-> StandardOutputs/Standard In Var 4
//     Standard Outputs/MAIN.R5.T02_CMD/SGs_ERRAck <-> StandardOutputs/Standard In Var 6
//     Standard Outputs/MAIN.R5.T02_CMD/SGs_RUNSTOP <-> StandardOutputs/Standard In Var 3
//     Standard Outputs/MAIN.R5.T02_CMD/SGs_RUNSTOP <-> StandardOutputs/Standard In Var 5
//     Standard Outputs/MAIN.Safety_Zone_Test <-> StandardOutputs/Standard In Var 21
//   SODG11_SSCC610_2403701_PLC/SODG11_SSCC610_2403701_PLC Instance <-> EtherCAT Master (EtherCAT)/R5.T01 (EK1100)/R5.T03 (EL1904)
//     Standard Inputs/MAIN.R5.T03/I <-> Module 1 (FSOES)/TxPDO/FSOE/InputChannel1
//     Standard Inputs/MAIN.R5.T03/I @bit 1 <-> Module 1 (FSOES)/TxPDO/FSOE/InputChannel2
//     Standard Inputs/MAIN.R5.T03/I @bit 2 <-> Module 1 (FSOES)/TxPDO/FSOE/InputChannel3
//     Standard Inputs/MAIN.R5.T03/I @bit 3 <-> Module 1 (FSOES)/TxPDO/FSOE/InputChannel4
//     Standard Inputs/MAIN.R5.T03/InfoData/State <-> InfoData/State
//   SODG11_SSCC610_2403701_PLC/SODG11_SSCC610_2403701_PLC Instance <-> EtherCAT Master (EtherCAT)/R5.T01 (EK1100)/R5.T04 (EK1122)
//     Standard Inputs/MAIN.R5.T04/InfoData/State <-> InfoData/State
//   SODG11_SSCC610_2403701_PLC/SODG11_SSCC610_2403701_PLC Instance <-> EtherCAT Master (EtherCAT)/R5.T01 (EK1100)/R5.T04 (EK1122)/R5.Reamer[1].N01 (EP1008-0002)
//     Standard Inputs/MAIN.R5.Reamer[1].N01/I <-> Channel 1/Input
//     Standard Inputs/MAIN.R5.Reamer[1].N01/I @bit 1 <-> Channel 2/Input
//     Standard Inputs/MAIN.R5.Reamer[1].N01/I @bit 2 <-> Channel 3/Input
//     Standard Inputs/MAIN.R5.Reamer[1].N01/I @bit 3 <-> Channel 4/Input
//     Standard Inputs/MAIN.R5.Reamer[1].N01/I @bit 4 <-> Channel 5/Input
//     Standard Inputs/MAIN.R5.Reamer[1].N01/I @bit 5 <-> Channel 6/Input
//     Standard Inputs/MAIN.R5.Reamer[1].N01/I @bit 6 <-> Channel 7/Input
//     Standard Inputs/MAIN.R5.Reamer[1].N01/I @bit 7 <-> Channel 8/Input
//     Standard Inputs/MAIN.R5.Reamer[1].N01/InfoData/State <-> InfoData/State
//     Standard Inputs/MAIN.R5.Reamer[1].N01/Wc_State <-> WcState/WcState
//   SODG11_SSCC610_2403701_PLC/SODG11_SSCC610_2403701_PLC Instance <-> EtherCAT Master (EtherCAT)/R5.T01 (EK1100)/R5.T04 (EK1122)/R5.Reamer[1].N30 (EP2028-0002)
//     Standard Inputs/MAIN.R5.Reamer[1].N30_STAT/InfoData/State <-> InfoData/State
//     Standard Outputs/MAIN.R5.Reamer[1].N30/Q <-> Channel 1/Output
//     Standard Outputs/MAIN.R5.Reamer[1].N30/Q @bit {1..7} <-> Channel {2..8}/Output  (7 links)
//   SODG11_SSCC610_2403701_PLC/SODG11_SSCC610_2403701_PLC Instance <-> EtherCAT Master (EtherCAT)/R6.RT02 (EL6695-1001)
//     Standard Inputs/MAIN.R6.In_From_HW/BYTE_[10] <-> Module 3 (Default IO)/Std. In (64 Bytes)/Input DWORD 2 @bit 8
//     Standard Inputs/MAIN.R6.In_From_HW/BYTE_[11] <-> Module 3 (Default IO)/Std. In (64 Bytes)/Input DWORD 2 @bit 16
//     Standard Inputs/MAIN.R6.In_From_HW/BYTE_[12] <-> Module 3 (Default IO)/Std. In (64 Bytes)/Input DWORD 2 @bit 24
//     Standard Inputs/MAIN.R6.In_From_HW/BYTE_[14] <-> Module 3 (Default IO)/Std. In (64 Bytes)/Input DWORD 3 @bit 8
//     Standard Inputs/MAIN.R6.In_From_HW/BYTE_[15] <-> Module 3 (Default IO)/Std. In (64 Bytes)/Input DWORD 3 @bit 16
//     Standard Inputs/MAIN.R6.In_From_HW/BYTE_[16] <-> Module 3 (Default IO)/Std. In (64 Bytes)/Input DWORD 3 @bit 24
//     Standard Inputs/MAIN.R6.In_From_HW/BYTE_[18] <-> Module 3 (Default IO)/Std. In (64 Bytes)/Input DWORD 4 @bit 8
//     Standard Inputs/MAIN.R6.In_From_HW/BYTE_[19] <-> Module 3 (Default IO)/Std. In (64 Bytes)/Input DWORD 4 @bit 16
//     Standard Inputs/MAIN.R6.In_From_HW/BYTE_[20] <-> Module 3 (Default IO)/Std. In (64 Bytes)/Input DWORD 4 @bit 24
//     Standard Inputs/MAIN.R6.In_From_HW/BYTE_[22] <-> Module 3 (Default IO)/Std. In (64 Bytes)/Input DWORD 5 @bit 8
//     Standard Inputs/MAIN.R6.In_From_HW/BYTE_[23] <-> Module 3 (Default IO)/Std. In (64 Bytes)/Input DWORD 5 @bit 16
//     Standard Inputs/MAIN.R6.In_From_HW/BYTE_[24] <-> Module 3 (Default IO)/Std. In (64 Bytes)/Input DWORD 5 @bit 24
//     Standard Inputs/MAIN.R6.In_From_HW/BYTE_[26] <-> Module 3 (Default IO)/Std. In (64 Bytes)/Input DWORD 6 @bit 8
//     Standard Inputs/MAIN.R6.In_From_HW/BYTE_[27] <-> Module 3 (Default IO)/Std. In (64 Bytes)/Input DWORD 6 @bit 16
//     Standard Inputs/MAIN.R6.In_From_HW/BYTE_[28] <-> Module 3 (Default IO)/Std. In (64 Bytes)/Input DWORD 6 @bit 24
//     Standard Inputs/MAIN.R6.In_From_HW/BYTE_[2] <-> Module 3 (Default IO)/Std. In (64 Bytes)/Input DWORD 0 @bit 8
//     Standard Inputs/MAIN.R6.In_From_HW/BYTE_[30] <-> Module 3 (Default IO)/Std. In (64 Bytes)/Input DWORD 7 @bit 8
//     Standard Inputs/MAIN.R6.In_From_HW/BYTE_[31] <-> Module 3 (Default IO)/Std. In (64 Bytes)/Input DWORD 7 @bit 16
//     Standard Inputs/MAIN.R6.In_From_HW/BYTE_[32] <-> Module 3 (Default IO)/Std. In (64 Bytes)/Input DWORD 7 @bit 24
//     Standard Inputs/MAIN.R6.In_From_HW/BYTE_[34] <-> Module 3 (Default IO)/Std. In (64 Bytes)/Input DWORD 8 @bit 8
//     Standard Inputs/MAIN.R6.In_From_HW/BYTE_[35] <-> Module 3 (Default IO)/Std. In (64 Bytes)/Input DWORD 8 @bit 16
//     Standard Inputs/MAIN.R6.In_From_HW/BYTE_[36] <-> Module 3 (Default IO)/Std. In (64 Bytes)/Input DWORD 8 @bit 24
//     Standard Inputs/MAIN.R6.In_From_HW/BYTE_[38] <-> Module 3 (Default IO)/Std. In (64 Bytes)/Input DWORD 9 @bit 8
//     Standard Inputs/MAIN.R6.In_From_HW/BYTE_[39] <-> Module 3 (Default IO)/Std. In (64 Bytes)/Input DWORD 9 @bit 16
//     Standard Inputs/MAIN.R6.In_From_HW/BYTE_[3] <-> Module 3 (Default IO)/Std. In (64 Bytes)/Input DWORD 0 @bit 16
//     Standard Inputs/MAIN.R6.In_From_HW/BYTE_[40] <-> Module 3 (Default IO)/Std. In (64 Bytes)/Input DWORD 9 @bit 24
//     Standard Inputs/MAIN.R6.In_From_HW/BYTE_[42] <-> Module 3 (Default IO)/Std. In (64 Bytes)/Input DWORD 10 @bit 8
//     Standard Inputs/MAIN.R6.In_From_HW/BYTE_[43] <-> Module 3 (Default IO)/Std. In (64 Bytes)/Input DWORD 10 @bit 16
//     Standard Inputs/MAIN.R6.In_From_HW/BYTE_[44] <-> Module 3 (Default IO)/Std. In (64 Bytes)/Input DWORD 10 @bit 24
//     Standard Inputs/MAIN.R6.In_From_HW/BYTE_[46] <-> Module 3 (Default IO)/Std. In (64 Bytes)/Input DWORD 11 @bit 8
//     Standard Inputs/MAIN.R6.In_From_HW/BYTE_[47] <-> Module 3 (Default IO)/Std. In (64 Bytes)/Input DWORD 11 @bit 16
//     Standard Inputs/MAIN.R6.In_From_HW/BYTE_[48] <-> Module 3 (Default IO)/Std. In (64 Bytes)/Input DWORD 11 @bit 24
//     Standard Inputs/MAIN.R6.In_From_HW/BYTE_[4] <-> Module 3 (Default IO)/Std. In (64 Bytes)/Input DWORD 0 @bit 24
//     Standard Inputs/MAIN.R6.In_From_HW/BYTE_[50] <-> Module 3 (Default IO)/Std. In (64 Bytes)/Input DWORD 12 @bit 8
//     Standard Inputs/MAIN.R6.In_From_HW/BYTE_[51] <-> Module 3 (Default IO)/Std. In (64 Bytes)/Input DWORD 12 @bit 16
//     Standard Inputs/MAIN.R6.In_From_HW/BYTE_[52] <-> Module 3 (Default IO)/Std. In (64 Bytes)/Input DWORD 12 @bit 24
//     Standard Inputs/MAIN.R6.In_From_HW/BYTE_[54] <-> Module 3 (Default IO)/Std. In (64 Bytes)/Input DWORD 13 @bit 8
//     Standard Inputs/MAIN.R6.In_From_HW/BYTE_[55] <-> Module 3 (Default IO)/Std. In (64 Bytes)/Input DWORD 13 @bit 16
//     Standard Inputs/MAIN.R6.In_From_HW/BYTE_[56] <-> Module 3 (Default IO)/Std. In (64 Bytes)/Input DWORD 13 @bit 24
//     Standard Inputs/MAIN.R6.In_From_HW/BYTE_[58] <-> Module 3 (Default IO)/Std. In (64 Bytes)/Input DWORD 14 @bit 8
//     Standard Inputs/MAIN.R6.In_From_HW/BYTE_[59] <-> Module 3 (Default IO)/Std. In (64 Bytes)/Input DWORD 14 @bit 16
//     Standard Inputs/MAIN.R6.In_From_HW/BYTE_[60] <-> Module 3 (Default IO)/Std. In (64 Bytes)/Input DWORD 14 @bit 24
//     Standard Inputs/MAIN.R6.In_From_HW/BYTE_[62] <-> Module 3 (Default IO)/Std. In (64 Bytes)/Input DWORD 15 @bit 8
//     Standard Inputs/MAIN.R6.In_From_HW/BYTE_[63] <-> Module 3 (Default IO)/Std. In (64 Bytes)/Input DWORD 15 @bit 16
//     Standard Inputs/MAIN.R6.In_From_HW/BYTE_[64] <-> Module 3 (Default IO)/Std. In (64 Bytes)/Input DWORD 15 @bit 24
//     Standard Inputs/MAIN.R6.In_From_HW/BYTE_[6] <-> Module 3 (Default IO)/Std. In (64 Bytes)/Input DWORD 1 @bit 8
//     Standard Inputs/MAIN.R6.In_From_HW/BYTE_[7] <-> Module 3 (Default IO)/Std. In (64 Bytes)/Input DWORD 1 @bit 16
//     Standard Inputs/MAIN.R6.In_From_HW/BYTE_[8] <-> Module 3 (Default IO)/Std. In (64 Bytes)/Input DWORD 1 @bit 24
//     Standard Inputs/MAIN.R6.In_From_HW/BYTE_[{1..61 step 4}] <-> Module 3 (Default IO)/Std. In (64 Bytes)/Input DWORD {0..15}  (16 links)
//     Standard Inputs/MAIN.R6.RT02/External_device_not_connected <-> Module 1 (Sync Inputs)/Compact/External device not connected
//     Standard Inputs/MAIN.R6.RT02/FSOE_Inputs_ConnID <-> Module 2 (Safety Data (8 Byte))/Inputs/FSOE/FSOE ConnID
//     Standard Inputs/MAIN.R6.RT02/FSOE_Inputs_Data_0 <-> Module 2 (Safety Data (8 Byte))/Inputs/FSOE/FSOE Data_0
//     Standard Inputs/MAIN.R6.RT02/FSOE_Inputs_Data_1 <-> Module 2 (Safety Data (8 Byte))/Inputs/FSOE/FSOE Data_1
//     Standard Inputs/MAIN.R6.RT02/FSOE_Inputs_Data_2 <-> Module 2 (Safety Data (8 Byte))/Inputs/FSOE/FSOE Data_2
//     Standard Inputs/MAIN.R6.RT02/FSOE_Inputs_Data_3 <-> Module 2 (Safety Data (8 Byte))/Inputs/FSOE/FSOE Data_3
//     Standard Inputs/MAIN.R6.RT02/InfoData/AdsAddr/netId <-> InfoData/AdsAddr/netId
//     Standard Inputs/MAIN.R6.RT02/InfoData/AdsAddr/port <-> InfoData/AdsAddr/port
//     Standard Inputs/MAIN.R6.RT02/InfoData/State <-> InfoData/State
//     Standard Inputs/MAIN.R6.RT02/TxPDO_State <-> Module 1 (Sync Inputs)/Compact/TxPDO state
//     Standard Inputs/MAIN.R6.RT02/TxPDO_Toogle <-> Module 1 (Sync Inputs)/Compact/TxPDO toggle
//     Standard Outputs/MAIN.R6.Out_To_HW/Byte_[10] <-> Module 3 (Default IO)/Std. Out (64 Bytes)/Output DWORD 2 @bit 8
//     Standard Outputs/MAIN.R6.Out_To_HW/Byte_[11] <-> Module 3 (Default IO)/Std. Out (64 Bytes)/Output DWORD 2 @bit 16
//     Standard Outputs/MAIN.R6.Out_To_HW/Byte_[12] <-> Module 3 (Default IO)/Std. Out (64 Bytes)/Output DWORD 2 @bit 24
//     Standard Outputs/MAIN.R6.Out_To_HW/Byte_[14] <-> Module 3 (Default IO)/Std. Out (64 Bytes)/Output DWORD 3 @bit 8
//     Standard Outputs/MAIN.R6.Out_To_HW/Byte_[15] <-> Module 3 (Default IO)/Std. Out (64 Bytes)/Output DWORD 3 @bit 16
//     Standard Outputs/MAIN.R6.Out_To_HW/Byte_[16] <-> Module 3 (Default IO)/Std. Out (64 Bytes)/Output DWORD 3 @bit 24
//     Standard Outputs/MAIN.R6.Out_To_HW/Byte_[18] <-> Module 3 (Default IO)/Std. Out (64 Bytes)/Output DWORD 4 @bit 8
//     Standard Outputs/MAIN.R6.Out_To_HW/Byte_[19] <-> Module 3 (Default IO)/Std. Out (64 Bytes)/Output DWORD 4 @bit 16
//     Standard Outputs/MAIN.R6.Out_To_HW/Byte_[20] <-> Module 3 (Default IO)/Std. Out (64 Bytes)/Output DWORD 4 @bit 24
//     Standard Outputs/MAIN.R6.Out_To_HW/Byte_[22] <-> Module 3 (Default IO)/Std. Out (64 Bytes)/Output DWORD 5 @bit 8
//     Standard Outputs/MAIN.R6.Out_To_HW/Byte_[23] <-> Module 3 (Default IO)/Std. Out (64 Bytes)/Output DWORD 5 @bit 16
//     Standard Outputs/MAIN.R6.Out_To_HW/Byte_[24] <-> Module 3 (Default IO)/Std. Out (64 Bytes)/Output DWORD 5 @bit 24
//     Standard Outputs/MAIN.R6.Out_To_HW/Byte_[26] <-> Module 3 (Default IO)/Std. Out (64 Bytes)/Output DWORD 6 @bit 8
//     Standard Outputs/MAIN.R6.Out_To_HW/Byte_[27] <-> Module 3 (Default IO)/Std. Out (64 Bytes)/Output DWORD 6 @bit 16
//     Standard Outputs/MAIN.R6.Out_To_HW/Byte_[28] <-> Module 3 (Default IO)/Std. Out (64 Bytes)/Output DWORD 6 @bit 24
//     Standard Outputs/MAIN.R6.Out_To_HW/Byte_[2] <-> Module 3 (Default IO)/Std. Out (64 Bytes)/Output DWORD 0 @bit 8
//     Standard Outputs/MAIN.R6.Out_To_HW/Byte_[30] <-> Module 3 (Default IO)/Std. Out (64 Bytes)/Output DWORD 7 @bit 8
//     Standard Outputs/MAIN.R6.Out_To_HW/Byte_[31] <-> Module 3 (Default IO)/Std. Out (64 Bytes)/Output DWORD 7 @bit 16
//     Standard Outputs/MAIN.R6.Out_To_HW/Byte_[32] <-> Module 3 (Default IO)/Std. Out (64 Bytes)/Output DWORD 7 @bit 24
//     Standard Outputs/MAIN.R6.Out_To_HW/Byte_[34] <-> Module 3 (Default IO)/Std. Out (64 Bytes)/Output DWORD 8 @bit 8
//     Standard Outputs/MAIN.R6.Out_To_HW/Byte_[35] <-> Module 3 (Default IO)/Std. Out (64 Bytes)/Output DWORD 8 @bit 16
//     Standard Outputs/MAIN.R6.Out_To_HW/Byte_[36] <-> Module 3 (Default IO)/Std. Out (64 Bytes)/Output DWORD 8 @bit 24
//     Standard Outputs/MAIN.R6.Out_To_HW/Byte_[38] <-> Module 3 (Default IO)/Std. Out (64 Bytes)/Output DWORD 9 @bit 8
//     Standard Outputs/MAIN.R6.Out_To_HW/Byte_[39] <-> Module 3 (Default IO)/Std. Out (64 Bytes)/Output DWORD 9 @bit 16
//     Standard Outputs/MAIN.R6.Out_To_HW/Byte_[3] <-> Module 3 (Default IO)/Std. Out (64 Bytes)/Output DWORD 0 @bit 16
//     Standard Outputs/MAIN.R6.Out_To_HW/Byte_[40] <-> Module 3 (Default IO)/Std. Out (64 Bytes)/Output DWORD 9 @bit 24
//     Standard Outputs/MAIN.R6.Out_To_HW/Byte_[42] <-> Module 3 (Default IO)/Std. Out (64 Bytes)/Output DWORD 10 @bit 8
//     Standard Outputs/MAIN.R6.Out_To_HW/Byte_[43] <-> Module 3 (Default IO)/Std. Out (64 Bytes)/Output DWORD 10 @bit 16
//     Standard Outputs/MAIN.R6.Out_To_HW/Byte_[44] <-> Module 3 (Default IO)/Std. Out (64 Bytes)/Output DWORD 10 @bit 24
//     Standard Outputs/MAIN.R6.Out_To_HW/Byte_[46] <-> Module 3 (Default IO)/Std. Out (64 Bytes)/Output DWORD 11 @bit 8
//     Standard Outputs/MAIN.R6.Out_To_HW/Byte_[47] <-> Module 3 (Default IO)/Std. Out (64 Bytes)/Output DWORD 11 @bit 16
//     Standard Outputs/MAIN.R6.Out_To_HW/Byte_[48] <-> Module 3 (Default IO)/Std. Out (64 Bytes)/Output DWORD 11 @bit 24
//     Standard Outputs/MAIN.R6.Out_To_HW/Byte_[4] <-> Module 3 (Default IO)/Std. Out (64 Bytes)/Output DWORD 0 @bit 24
//     Standard Outputs/MAIN.R6.Out_To_HW/Byte_[50] <-> Module 3 (Default IO)/Std. Out (64 Bytes)/Output DWORD 12 @bit 8
//     Standard Outputs/MAIN.R6.Out_To_HW/Byte_[51] <-> Module 3 (Default IO)/Std. Out (64 Bytes)/Output DWORD 12 @bit 16
//     Standard Outputs/MAIN.R6.Out_To_HW/Byte_[52] <-> Module 3 (Default IO)/Std. Out (64 Bytes)/Output DWORD 12 @bit 24
//     Standard Outputs/MAIN.R6.Out_To_HW/Byte_[54] <-> Module 3 (Default IO)/Std. Out (64 Bytes)/Output DWORD 13 @bit 8
//     Standard Outputs/MAIN.R6.Out_To_HW/Byte_[55] <-> Module 3 (Default IO)/Std. Out (64 Bytes)/Output DWORD 13 @bit 16
//     Standard Outputs/MAIN.R6.Out_To_HW/Byte_[56] <-> Module 3 (Default IO)/Std. Out (64 Bytes)/Output DWORD 13 @bit 24
//     Standard Outputs/MAIN.R6.Out_To_HW/Byte_[58] <-> Module 3 (Default IO)/Std. Out (64 Bytes)/Output DWORD 14 @bit 8
//     Standard Outputs/MAIN.R6.Out_To_HW/Byte_[59] <-> Module 3 (Default IO)/Std. Out (64 Bytes)/Output DWORD 14 @bit 16
//     Standard Outputs/MAIN.R6.Out_To_HW/Byte_[60] <-> Module 3 (Default IO)/Std. Out (64 Bytes)/Output DWORD 14 @bit 24
//     Standard Outputs/MAIN.R6.Out_To_HW/Byte_[62] <-> Module 3 (Default IO)/Std. Out (64 Bytes)/Output DWORD 15 @bit 8
//     Standard Outputs/MAIN.R6.Out_To_HW/Byte_[63] <-> Module 3 (Default IO)/Std. Out (64 Bytes)/Output DWORD 15 @bit 16
//     Standard Outputs/MAIN.R6.Out_To_HW/Byte_[64] <-> Module 3 (Default IO)/Std. Out (64 Bytes)/Output DWORD 15 @bit 24
//     Standard Outputs/MAIN.R6.Out_To_HW/Byte_[6] <-> Module 3 (Default IO)/Std. Out (64 Bytes)/Output DWORD 1 @bit 8
//     Standard Outputs/MAIN.R6.Out_To_HW/Byte_[7] <-> Module 3 (Default IO)/Std. Out (64 Bytes)/Output DWORD 1 @bit 16
//     Standard Outputs/MAIN.R6.Out_To_HW/Byte_[8] <-> Module 3 (Default IO)/Std. Out (64 Bytes)/Output DWORD 1 @bit 24
//     Standard Outputs/MAIN.R6.Out_To_HW/Byte_[{1..61 step 4}] <-> Module 3 (Default IO)/Std. Out (64 Bytes)/Output DWORD {0..15}  (16 links)
//   SODG11_SSCC610_2403701_PLC/SODG11_SSCC610_2403701_PLC Instance <-> EtherCAT Master (EtherCAT)/R6.T01 (EK1100)
//     Standard Inputs/MAIN.R6.T01/InfoData/State <-> InfoData/State
//   SODG11_SSCC610_2403701_PLC/SODG11_SSCC610_2403701_PLC Instance <-> EtherCAT Master (EtherCAT)/R6.T01 (EK1100)/R6.T02 (EL6900)
//     Standard Inputs/MAIN.R6.RT02/FSOE_Outputs_Data_0 @bit 1 <-> StandardInputs/Standard Out Var 14
//     Standard Inputs/MAIN.R6.RT02/FSOE_Outputs_Data_0 @bit 2 <-> StandardInputs/Standard Out Var 15
//     Standard Inputs/MAIN.R6.RT02/FSOE_Outputs_Data_2 @bit 1 <-> StandardInputs/Standard Out Var 18
//     Standard Inputs/MAIN.R6.RT02/FSOE_Outputs_Data_2 <-> StandardInputs/Standard Out Var 17
//     Standard Inputs/MAIN.R6.T02_STAT/Device_Info_Data/Project_CRC <-> Device Info Data/Project CRC
//     Standard Inputs/MAIN.R6.T02_STAT/FBs_FB_ERR <-> StandardInputs/Standard Out Var 16
//     Standard Inputs/MAIN.R6.T02_STAT/FBs_FB_ERR @bit 16 <-> StandardInputs/Standard Out Var 19
//     Standard Inputs/MAIN.R6.T02_STAT/FBs_FB_ERR @bit 29 <-> StandardInputs/Standard Out Var 20
//     Standard Inputs/MAIN.R6.T02_STAT/InfoData/AdsAddr/netId <-> InfoData/AdsAddr/netId
//     Standard Inputs/MAIN.R6.T02_STAT/InfoData/AdsAddr/port <-> InfoData/AdsAddr/port
//     Standard Inputs/MAIN.R6.T02_STAT/InfoData/State <-> InfoData/State
//     Standard Inputs/MAIN.R6.T02_STAT/SGs_COM_ERR @bit 1 <-> StandardInputs/Standard Out Var 12
//     Standard Inputs/MAIN.R6.T02_STAT/SGs_COM_ERR <-> StandardInputs/Standard Out Var 9
//     Standard Inputs/MAIN.R6.T02_STAT/SGs_FB_ERR @bit 1 <-> StandardInputs/Standard Out Var 11
//     Standard Inputs/MAIN.R6.T02_STAT/SGs_FB_ERR <-> StandardInputs/Standard Out Var 8
//     Standard Inputs/MAIN.R6.T02_STAT/SGs_OUT_ERR <-> StandardInputs/Standard Out Var 10
//     Standard Inputs/MAIN.R6.T02_STAT/SGs_OUT_ERR @bit 1 <-> StandardInputs/Standard Out Var 13
//     Standard Outputs/MAIN.R6.T02_CMD/FBs_ControlPowerPB <-> StandardOutputs/Standard In Var 7
//     Standard Outputs/MAIN.R6.T02_CMD/SGs_ERRAck <-> StandardOutputs/Standard In Var 4
//     Standard Outputs/MAIN.R6.T02_CMD/SGs_ERRAck <-> StandardOutputs/Standard In Var 6
//     Standard Outputs/MAIN.R6.T02_CMD/SGs_RUNSTOP <-> StandardOutputs/Standard In Var 3
//     Standard Outputs/MAIN.R6.T02_CMD/SGs_RUNSTOP <-> StandardOutputs/Standard In Var 5
//     Standard Outputs/MAIN.Safety_Zone_Test <-> StandardOutputs/Standard In Var 21
//   SODG11_SSCC610_2403701_PLC/SODG11_SSCC610_2403701_PLC Instance <-> EtherCAT Master (EtherCAT)/R6.T01 (EK1100)/R6.T03 (EL1904)
//     Standard Inputs/MAIN.R6.T03/I <-> Module 1 (FSOES)/TxPDO/FSOE/InputChannel1
//     Standard Inputs/MAIN.R6.T03/I @bit 1 <-> Module 1 (FSOES)/TxPDO/FSOE/InputChannel2
//     Standard Inputs/MAIN.R6.T03/I @bit 2 <-> Module 1 (FSOES)/TxPDO/FSOE/InputChannel3
//     Standard Inputs/MAIN.R6.T03/I @bit 3 <-> Module 1 (FSOES)/TxPDO/FSOE/InputChannel4
//     Standard Inputs/MAIN.R6.T03/InfoData/State <-> InfoData/State
//   SODG11_SSCC610_2403701_PLC/SODG11_SSCC610_2403701_PLC Instance <-> EtherCAT Master (EtherCAT)/R6.T01 (EK1100)/R6.T04 (EK1122)
//     Standard Inputs/MAIN.R6.T04/InfoData/State <-> InfoData/State
//   SODG11_SSCC610_2403701_PLC/SODG11_SSCC610_2403701_PLC Instance <-> EtherCAT Master (EtherCAT)/R6.T01 (EK1100)/R6.T04 (EK1122)/R6.Reamer[1].N01 (EP1008-0002)
//     Standard Inputs/MAIN.R6.Reamer[1].N01/I <-> Channel 1/Input
//     Standard Inputs/MAIN.R6.Reamer[1].N01/I @bit 1 <-> Channel 2/Input
//     Standard Inputs/MAIN.R6.Reamer[1].N01/I @bit 2 <-> Channel 3/Input
//     Standard Inputs/MAIN.R6.Reamer[1].N01/I @bit 3 <-> Channel 4/Input
//     Standard Inputs/MAIN.R6.Reamer[1].N01/I @bit 4 <-> Channel 5/Input
//     Standard Inputs/MAIN.R6.Reamer[1].N01/I @bit 5 <-> Channel 6/Input
//     Standard Inputs/MAIN.R6.Reamer[1].N01/I @bit 6 <-> Channel 7/Input
//     Standard Inputs/MAIN.R6.Reamer[1].N01/I @bit 7 <-> Channel 8/Input
//     Standard Inputs/MAIN.R6.Reamer[1].N01/InfoData/State <-> InfoData/State
//     Standard Inputs/MAIN.R6.Reamer[1].N01/Wc_State <-> WcState/WcState
//   SODG11_SSCC610_2403701_PLC/SODG11_SSCC610_2403701_PLC Instance <-> EtherCAT Master (EtherCAT)/R6.T01 (EK1100)/R6.T04 (EK1122)/R6.Reamer[1].N30 (EP2028-0002)
//     Standard Inputs/MAIN.R6.Reamer[1].N30_STAT/InfoData/State <-> InfoData/State
//     Standard Outputs/MAIN.R6.Reamer[1].N30/Q <-> Channel 1/Output
//     Standard Outputs/MAIN.R6.Reamer[1].N30/Q @bit {1..7} <-> Channel {2..8}/Output  (7 links)
//   SODG11_SSCC610_2403701_PLC/SODG11_SSCC610_2403701_PLC Instance <-> EtherCAT Master (EtherCAT)/R7.RT02 (EL6695-1001)
//     Standard Inputs/MAIN.R7.In_From_HW/BYTE_[10] <-> Module 3 (Default IO)/Std. In (64 Bytes)/Input DWORD 2 @bit 8
//     Standard Inputs/MAIN.R7.In_From_HW/BYTE_[11] <-> Module 3 (Default IO)/Std. In (64 Bytes)/Input DWORD 2 @bit 16
//     Standard Inputs/MAIN.R7.In_From_HW/BYTE_[12] <-> Module 3 (Default IO)/Std. In (64 Bytes)/Input DWORD 2 @bit 24
//     Standard Inputs/MAIN.R7.In_From_HW/BYTE_[14] <-> Module 3 (Default IO)/Std. In (64 Bytes)/Input DWORD 3 @bit 8
//     Standard Inputs/MAIN.R7.In_From_HW/BYTE_[15] <-> Module 3 (Default IO)/Std. In (64 Bytes)/Input DWORD 3 @bit 16
//     Standard Inputs/MAIN.R7.In_From_HW/BYTE_[16] <-> Module 3 (Default IO)/Std. In (64 Bytes)/Input DWORD 3 @bit 24
//     Standard Inputs/MAIN.R7.In_From_HW/BYTE_[18] <-> Module 3 (Default IO)/Std. In (64 Bytes)/Input DWORD 4 @bit 8
//     Standard Inputs/MAIN.R7.In_From_HW/BYTE_[19] <-> Module 3 (Default IO)/Std. In (64 Bytes)/Input DWORD 4 @bit 16
//     Standard Inputs/MAIN.R7.In_From_HW/BYTE_[20] <-> Module 3 (Default IO)/Std. In (64 Bytes)/Input DWORD 4 @bit 24
//     Standard Inputs/MAIN.R7.In_From_HW/BYTE_[22] <-> Module 3 (Default IO)/Std. In (64 Bytes)/Input DWORD 5 @bit 8
//     Standard Inputs/MAIN.R7.In_From_HW/BYTE_[23] <-> Module 3 (Default IO)/Std. In (64 Bytes)/Input DWORD 5 @bit 16
//     Standard Inputs/MAIN.R7.In_From_HW/BYTE_[24] <-> Module 3 (Default IO)/Std. In (64 Bytes)/Input DWORD 5 @bit 24
//     Standard Inputs/MAIN.R7.In_From_HW/BYTE_[26] <-> Module 3 (Default IO)/Std. In (64 Bytes)/Input DWORD 6 @bit 8
//     Standard Inputs/MAIN.R7.In_From_HW/BYTE_[27] <-> Module 3 (Default IO)/Std. In (64 Bytes)/Input DWORD 6 @bit 16
//     Standard Inputs/MAIN.R7.In_From_HW/BYTE_[28] <-> Module 3 (Default IO)/Std. In (64 Bytes)/Input DWORD 6 @bit 24
//     Standard Inputs/MAIN.R7.In_From_HW/BYTE_[2] <-> Module 3 (Default IO)/Std. In (64 Bytes)/Input DWORD 0 @bit 8
//     Standard Inputs/MAIN.R7.In_From_HW/BYTE_[30] <-> Module 3 (Default IO)/Std. In (64 Bytes)/Input DWORD 7 @bit 8
//     Standard Inputs/MAIN.R7.In_From_HW/BYTE_[31] <-> Module 3 (Default IO)/Std. In (64 Bytes)/Input DWORD 7 @bit 16
//     Standard Inputs/MAIN.R7.In_From_HW/BYTE_[32] <-> Module 3 (Default IO)/Std. In (64 Bytes)/Input DWORD 7 @bit 24
//     Standard Inputs/MAIN.R7.In_From_HW/BYTE_[34] <-> Module 3 (Default IO)/Std. In (64 Bytes)/Input DWORD 8 @bit 8
//     Standard Inputs/MAIN.R7.In_From_HW/BYTE_[35] <-> Module 3 (Default IO)/Std. In (64 Bytes)/Input DWORD 8 @bit 16
//     Standard Inputs/MAIN.R7.In_From_HW/BYTE_[36] <-> Module 3 (Default IO)/Std. In (64 Bytes)/Input DWORD 8 @bit 24
//     Standard Inputs/MAIN.R7.In_From_HW/BYTE_[38] <-> Module 3 (Default IO)/Std. In (64 Bytes)/Input DWORD 9 @bit 8
//     Standard Inputs/MAIN.R7.In_From_HW/BYTE_[39] <-> Module 3 (Default IO)/Std. In (64 Bytes)/Input DWORD 9 @bit 16
//     Standard Inputs/MAIN.R7.In_From_HW/BYTE_[3] <-> Module 3 (Default IO)/Std. In (64 Bytes)/Input DWORD 0 @bit 16
//     Standard Inputs/MAIN.R7.In_From_HW/BYTE_[40] <-> Module 3 (Default IO)/Std. In (64 Bytes)/Input DWORD 9 @bit 24
//     Standard Inputs/MAIN.R7.In_From_HW/BYTE_[42] <-> Module 3 (Default IO)/Std. In (64 Bytes)/Input DWORD 10 @bit 8
//     Standard Inputs/MAIN.R7.In_From_HW/BYTE_[43] <-> Module 3 (Default IO)/Std. In (64 Bytes)/Input DWORD 10 @bit 16
//     Standard Inputs/MAIN.R7.In_From_HW/BYTE_[44] <-> Module 3 (Default IO)/Std. In (64 Bytes)/Input DWORD 10 @bit 24
//     Standard Inputs/MAIN.R7.In_From_HW/BYTE_[46] <-> Module 3 (Default IO)/Std. In (64 Bytes)/Input DWORD 11 @bit 8
//     Standard Inputs/MAIN.R7.In_From_HW/BYTE_[47] <-> Module 3 (Default IO)/Std. In (64 Bytes)/Input DWORD 11 @bit 16
//     Standard Inputs/MAIN.R7.In_From_HW/BYTE_[48] <-> Module 3 (Default IO)/Std. In (64 Bytes)/Input DWORD 11 @bit 24
//     Standard Inputs/MAIN.R7.In_From_HW/BYTE_[4] <-> Module 3 (Default IO)/Std. In (64 Bytes)/Input DWORD 0 @bit 24
//     Standard Inputs/MAIN.R7.In_From_HW/BYTE_[50] <-> Module 3 (Default IO)/Std. In (64 Bytes)/Input DWORD 12 @bit 8
//     Standard Inputs/MAIN.R7.In_From_HW/BYTE_[51] <-> Module 3 (Default IO)/Std. In (64 Bytes)/Input DWORD 12 @bit 16
//     Standard Inputs/MAIN.R7.In_From_HW/BYTE_[52] <-> Module 3 (Default IO)/Std. In (64 Bytes)/Input DWORD 12 @bit 24
//     Standard Inputs/MAIN.R7.In_From_HW/BYTE_[54] <-> Module 3 (Default IO)/Std. In (64 Bytes)/Input DWORD 13 @bit 8
//     Standard Inputs/MAIN.R7.In_From_HW/BYTE_[55] <-> Module 3 (Default IO)/Std. In (64 Bytes)/Input DWORD 13 @bit 16
//     Standard Inputs/MAIN.R7.In_From_HW/BYTE_[56] <-> Module 3 (Default IO)/Std. In (64 Bytes)/Input DWORD 13 @bit 24
//     Standard Inputs/MAIN.R7.In_From_HW/BYTE_[58] <-> Module 3 (Default IO)/Std. In (64 Bytes)/Input DWORD 14 @bit 8
//     Standard Inputs/MAIN.R7.In_From_HW/BYTE_[59] <-> Module 3 (Default IO)/Std. In (64 Bytes)/Input DWORD 14 @bit 16
//     Standard Inputs/MAIN.R7.In_From_HW/BYTE_[60] <-> Module 3 (Default IO)/Std. In (64 Bytes)/Input DWORD 14 @bit 24
//     Standard Inputs/MAIN.R7.In_From_HW/BYTE_[62] <-> Module 3 (Default IO)/Std. In (64 Bytes)/Input DWORD 15 @bit 8
//     Standard Inputs/MAIN.R7.In_From_HW/BYTE_[63] <-> Module 3 (Default IO)/Std. In (64 Bytes)/Input DWORD 15 @bit 16
//     Standard Inputs/MAIN.R7.In_From_HW/BYTE_[64] <-> Module 3 (Default IO)/Std. In (64 Bytes)/Input DWORD 15 @bit 24
//     Standard Inputs/MAIN.R7.In_From_HW/BYTE_[6] <-> Module 3 (Default IO)/Std. In (64 Bytes)/Input DWORD 1 @bit 8
//     Standard Inputs/MAIN.R7.In_From_HW/BYTE_[7] <-> Module 3 (Default IO)/Std. In (64 Bytes)/Input DWORD 1 @bit 16
//     Standard Inputs/MAIN.R7.In_From_HW/BYTE_[8] <-> Module 3 (Default IO)/Std. In (64 Bytes)/Input DWORD 1 @bit 24
//     Standard Inputs/MAIN.R7.In_From_HW/BYTE_[{1..61 step 4}] <-> Module 3 (Default IO)/Std. In (64 Bytes)/Input DWORD {0..15}  (16 links)
//     Standard Inputs/MAIN.R7.RT02/External_device_not_connected <-> Module 1 (Sync Inputs)/Compact/External device not connected
//     Standard Inputs/MAIN.R7.RT02/FSOE_Inputs_ConnID <-> Module 2 (Safety Data (8 Byte))/Inputs/FSOE/FSOE ConnID
//     Standard Inputs/MAIN.R7.RT02/FSOE_Inputs_Data_0 <-> Module 2 (Safety Data (8 Byte))/Inputs/FSOE/FSOE Data_0
//     Standard Inputs/MAIN.R7.RT02/FSOE_Inputs_Data_1 <-> Module 2 (Safety Data (8 Byte))/Inputs/FSOE/FSOE Data_1
//     Standard Inputs/MAIN.R7.RT02/FSOE_Inputs_Data_2 <-> Module 2 (Safety Data (8 Byte))/Inputs/FSOE/FSOE Data_2
//     Standard Inputs/MAIN.R7.RT02/FSOE_Inputs_Data_3 <-> Module 2 (Safety Data (8 Byte))/Inputs/FSOE/FSOE Data_3
//     Standard Inputs/MAIN.R7.RT02/InfoData/AdsAddr/netId <-> InfoData/AdsAddr/netId
//     Standard Inputs/MAIN.R7.RT02/InfoData/AdsAddr/port <-> InfoData/AdsAddr/port
//     Standard Inputs/MAIN.R7.RT02/InfoData/State <-> InfoData/State
//     Standard Inputs/MAIN.R7.RT02/TxPDO_State <-> Module 1 (Sync Inputs)/Compact/TxPDO state
//     Standard Inputs/MAIN.R7.RT02/TxPDO_Toogle <-> Module 1 (Sync Inputs)/Compact/TxPDO toggle
//     Standard Outputs/MAIN.R7.Out_To_HW/Byte_[10] <-> Module 3 (Default IO)/Std. Out (64 Bytes)/Output DWORD 2 @bit 8
//     Standard Outputs/MAIN.R7.Out_To_HW/Byte_[11] <-> Module 3 (Default IO)/Std. Out (64 Bytes)/Output DWORD 2 @bit 16
//     Standard Outputs/MAIN.R7.Out_To_HW/Byte_[12] <-> Module 3 (Default IO)/Std. Out (64 Bytes)/Output DWORD 2 @bit 24
//     Standard Outputs/MAIN.R7.Out_To_HW/Byte_[14] <-> Module 3 (Default IO)/Std. Out (64 Bytes)/Output DWORD 3 @bit 8
//     Standard Outputs/MAIN.R7.Out_To_HW/Byte_[15] <-> Module 3 (Default IO)/Std. Out (64 Bytes)/Output DWORD 3 @bit 16
//     Standard Outputs/MAIN.R7.Out_To_HW/Byte_[16] <-> Module 3 (Default IO)/Std. Out (64 Bytes)/Output DWORD 3 @bit 24
//     Standard Outputs/MAIN.R7.Out_To_HW/Byte_[18] <-> Module 3 (Default IO)/Std. Out (64 Bytes)/Output DWORD 4 @bit 8
//     Standard Outputs/MAIN.R7.Out_To_HW/Byte_[19] <-> Module 3 (Default IO)/Std. Out (64 Bytes)/Output DWORD 4 @bit 16
//     Standard Outputs/MAIN.R7.Out_To_HW/Byte_[20] <-> Module 3 (Default IO)/Std. Out (64 Bytes)/Output DWORD 4 @bit 24
//     Standard Outputs/MAIN.R7.Out_To_HW/Byte_[22] <-> Module 3 (Default IO)/Std. Out (64 Bytes)/Output DWORD 5 @bit 8
//     Standard Outputs/MAIN.R7.Out_To_HW/Byte_[23] <-> Module 3 (Default IO)/Std. Out (64 Bytes)/Output DWORD 5 @bit 16
//     Standard Outputs/MAIN.R7.Out_To_HW/Byte_[24] <-> Module 3 (Default IO)/Std. Out (64 Bytes)/Output DWORD 5 @bit 24
//     Standard Outputs/MAIN.R7.Out_To_HW/Byte_[26] <-> Module 3 (Default IO)/Std. Out (64 Bytes)/Output DWORD 6 @bit 8
//     Standard Outputs/MAIN.R7.Out_To_HW/Byte_[27] <-> Module 3 (Default IO)/Std. Out (64 Bytes)/Output DWORD 6 @bit 16
//     Standard Outputs/MAIN.R7.Out_To_HW/Byte_[28] <-> Module 3 (Default IO)/Std. Out (64 Bytes)/Output DWORD 6 @bit 24
//     Standard Outputs/MAIN.R7.Out_To_HW/Byte_[2] <-> Module 3 (Default IO)/Std. Out (64 Bytes)/Output DWORD 0 @bit 8
//     Standard Outputs/MAIN.R7.Out_To_HW/Byte_[30] <-> Module 3 (Default IO)/Std. Out (64 Bytes)/Output DWORD 7 @bit 8
//     Standard Outputs/MAIN.R7.Out_To_HW/Byte_[31] <-> Module 3 (Default IO)/Std. Out (64 Bytes)/Output DWORD 7 @bit 16
//     Standard Outputs/MAIN.R7.Out_To_HW/Byte_[32] <-> Module 3 (Default IO)/Std. Out (64 Bytes)/Output DWORD 7 @bit 24
//     Standard Outputs/MAIN.R7.Out_To_HW/Byte_[34] <-> Module 3 (Default IO)/Std. Out (64 Bytes)/Output DWORD 8 @bit 8
//     Standard Outputs/MAIN.R7.Out_To_HW/Byte_[35] <-> Module 3 (Default IO)/Std. Out (64 Bytes)/Output DWORD 8 @bit 16
//     Standard Outputs/MAIN.R7.Out_To_HW/Byte_[36] <-> Module 3 (Default IO)/Std. Out (64 Bytes)/Output DWORD 8 @bit 24
//     Standard Outputs/MAIN.R7.Out_To_HW/Byte_[38] <-> Module 3 (Default IO)/Std. Out (64 Bytes)/Output DWORD 9 @bit 8
//     Standard Outputs/MAIN.R7.Out_To_HW/Byte_[39] <-> Module 3 (Default IO)/Std. Out (64 Bytes)/Output DWORD 9 @bit 16
//     Standard Outputs/MAIN.R7.Out_To_HW/Byte_[3] <-> Module 3 (Default IO)/Std. Out (64 Bytes)/Output DWORD 0 @bit 16
//     Standard Outputs/MAIN.R7.Out_To_HW/Byte_[40] <-> Module 3 (Default IO)/Std. Out (64 Bytes)/Output DWORD 9 @bit 24
//     Standard Outputs/MAIN.R7.Out_To_HW/Byte_[42] <-> Module 3 (Default IO)/Std. Out (64 Bytes)/Output DWORD 10 @bit 8
//     Standard Outputs/MAIN.R7.Out_To_HW/Byte_[43] <-> Module 3 (Default IO)/Std. Out (64 Bytes)/Output DWORD 10 @bit 16
//     Standard Outputs/MAIN.R7.Out_To_HW/Byte_[44] <-> Module 3 (Default IO)/Std. Out (64 Bytes)/Output DWORD 10 @bit 24
//     Standard Outputs/MAIN.R7.Out_To_HW/Byte_[46] <-> Module 3 (Default IO)/Std. Out (64 Bytes)/Output DWORD 11 @bit 8
//     Standard Outputs/MAIN.R7.Out_To_HW/Byte_[47] <-> Module 3 (Default IO)/Std. Out (64 Bytes)/Output DWORD 11 @bit 16
//     Standard Outputs/MAIN.R7.Out_To_HW/Byte_[48] <-> Module 3 (Default IO)/Std. Out (64 Bytes)/Output DWORD 11 @bit 24
//     Standard Outputs/MAIN.R7.Out_To_HW/Byte_[4] <-> Module 3 (Default IO)/Std. Out (64 Bytes)/Output DWORD 0 @bit 24
//     Standard Outputs/MAIN.R7.Out_To_HW/Byte_[50] <-> Module 3 (Default IO)/Std. Out (64 Bytes)/Output DWORD 12 @bit 8
//     Standard Outputs/MAIN.R7.Out_To_HW/Byte_[51] <-> Module 3 (Default IO)/Std. Out (64 Bytes)/Output DWORD 12 @bit 16
//     Standard Outputs/MAIN.R7.Out_To_HW/Byte_[52] <-> Module 3 (Default IO)/Std. Out (64 Bytes)/Output DWORD 12 @bit 24
//     Standard Outputs/MAIN.R7.Out_To_HW/Byte_[54] <-> Module 3 (Default IO)/Std. Out (64 Bytes)/Output DWORD 13 @bit 8
//     Standard Outputs/MAIN.R7.Out_To_HW/Byte_[55] <-> Module 3 (Default IO)/Std. Out (64 Bytes)/Output DWORD 13 @bit 16
//     Standard Outputs/MAIN.R7.Out_To_HW/Byte_[56] <-> Module 3 (Default IO)/Std. Out (64 Bytes)/Output DWORD 13 @bit 24
//     Standard Outputs/MAIN.R7.Out_To_HW/Byte_[58] <-> Module 3 (Default IO)/Std. Out (64 Bytes)/Output DWORD 14 @bit 8
//     Standard Outputs/MAIN.R7.Out_To_HW/Byte_[59] <-> Module 3 (Default IO)/Std. Out (64 Bytes)/Output DWORD 14 @bit 16
//     Standard Outputs/MAIN.R7.Out_To_HW/Byte_[60] <-> Module 3 (Default IO)/Std. Out (64 Bytes)/Output DWORD 14 @bit 24
//     Standard Outputs/MAIN.R7.Out_To_HW/Byte_[62] <-> Module 3 (Default IO)/Std. Out (64 Bytes)/Output DWORD 15 @bit 8
//     Standard Outputs/MAIN.R7.Out_To_HW/Byte_[63] <-> Module 3 (Default IO)/Std. Out (64 Bytes)/Output DWORD 15 @bit 16
//     Standard Outputs/MAIN.R7.Out_To_HW/Byte_[64] <-> Module 3 (Default IO)/Std. Out (64 Bytes)/Output DWORD 15 @bit 24
//     Standard Outputs/MAIN.R7.Out_To_HW/Byte_[6] <-> Module 3 (Default IO)/Std. Out (64 Bytes)/Output DWORD 1 @bit 8
//     Standard Outputs/MAIN.R7.Out_To_HW/Byte_[7] <-> Module 3 (Default IO)/Std. Out (64 Bytes)/Output DWORD 1 @bit 16
//     Standard Outputs/MAIN.R7.Out_To_HW/Byte_[8] <-> Module 3 (Default IO)/Std. Out (64 Bytes)/Output DWORD 1 @bit 24
//     Standard Outputs/MAIN.R7.Out_To_HW/Byte_[{1..61 step 4}] <-> Module 3 (Default IO)/Std. Out (64 Bytes)/Output DWORD {0..15}  (16 links)
//   SODG11_SSCC610_2403701_PLC/SODG11_SSCC610_2403701_PLC Instance <-> EtherCAT Master (EtherCAT)/R7.T01 (EK1100)
//     Standard Inputs/MAIN.R7.T01/InfoData/State <-> InfoData/State
//   SODG11_SSCC610_2403701_PLC/SODG11_SSCC610_2403701_PLC Instance <-> EtherCAT Master (EtherCAT)/R7.T01 (EK1100)/R7.T02 (EL6900)
//     Standard Inputs/MAIN.R7.RT02/FSOE_Outputs_Data_0 @bit 1 <-> StandardInputs/Standard Out Var 14
//     Standard Inputs/MAIN.R7.RT02/FSOE_Outputs_Data_0 @bit 2 <-> StandardInputs/Standard Out Var 15
//     Standard Inputs/MAIN.R7.RT02/FSOE_Outputs_Data_2 @bit 1 <-> StandardInputs/Standard Out Var 18
//     Standard Inputs/MAIN.R7.RT02/FSOE_Outputs_Data_2 <-> StandardInputs/Standard Out Var 17
//     Standard Inputs/MAIN.R7.T02_STAT/Device_Info_Data/Project_CRC <-> Device Info Data/Project CRC
//     Standard Inputs/MAIN.R7.T02_STAT/FBs_FB_ERR <-> StandardInputs/Standard Out Var 16
//     Standard Inputs/MAIN.R7.T02_STAT/FBs_FB_ERR @bit 16 <-> StandardInputs/Standard Out Var 19
//     Standard Inputs/MAIN.R7.T02_STAT/FBs_FB_ERR @bit 29 <-> StandardInputs/Standard Out Var 20
//     Standard Inputs/MAIN.R7.T02_STAT/InfoData/AdsAddr/netId <-> InfoData/AdsAddr/netId
//     Standard Inputs/MAIN.R7.T02_STAT/InfoData/AdsAddr/port <-> InfoData/AdsAddr/port
//     Standard Inputs/MAIN.R7.T02_STAT/InfoData/State <-> InfoData/State
